Universal Robots URScript: Step Corner Extended.script

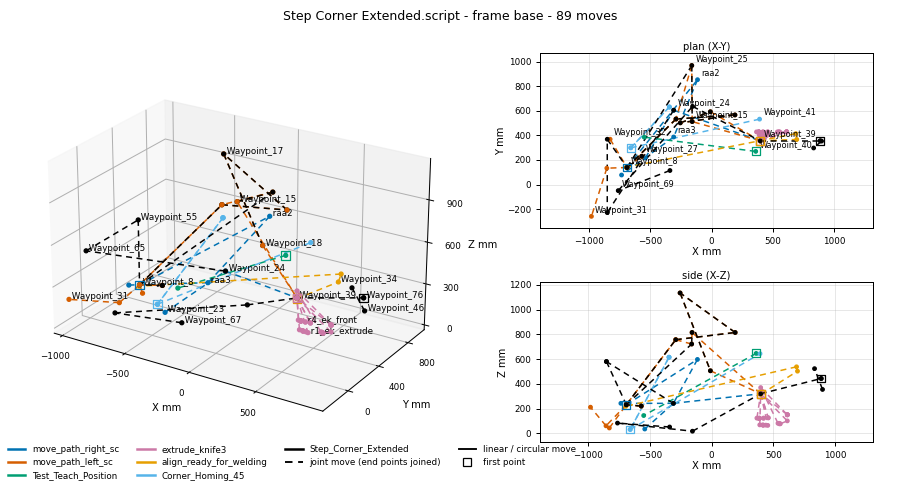
[picture p0: tool path of Step Corner Extended.script in frame base, 89 of 174 moves have a stored position in this frame; points joined in program order, loops and branches not executed]
def Step_Corner_Extended():
  global _hidden_verificationVariable=0
  set_standard_analog_input_domain(0, 1)
  set_standard_analog_input_domain(1, 1)
  set_tool_analog_input_domain(0, 1)
  set_tool_analog_input_domain(1, 1)
  set_analog_outputdomain(0, 0)
  set_analog_outputdomain(1, 0)
  set_input_actions_to_default()
  set_target_payload(10.800000, [-0.001000, -0.053000, 0.068000], [0.081228, 0.081228, 0.081228, 0.000000, 0.000000, 0.000000])
  set_tool_communication(False, 115200, 0, 1, 1.5, 3.5)
  set_tool_output_mode(0)
  set_tool_digital_output_mode(0, 1)
  set_tool_digital_output_mode(1, 1)
  set_tool_voltage(0)
  set_tcp(p[-0.011699999999999999,-0.328,0.105,1.2092,-1.2092,1.2092])
  set_safety_mode_transition_hardness(1)
  set_gravity([0.0, 0.0, 9.82])
  global robot_number=3
  global Point_1=p[0.0,0.0,0.0,0.0,0.0,0.0]
  global Point_2=p[0.0,0.0,0.0,0.0,0.0,0.0]
  # begin: URCap Installation Node
  #   Source: UR Connect, 1.13.79, Universal Robots
  #   Type: UR Connect
  myurRPC = rpc_factory("xmlrpc","http://127.0.0.1:40474")
  # end: URCap Installation Node
  # begin: URCap Installation Node
  #   Source: MachineLogic for Universal Robots, 3.1.7, Vention Inc.
  #   Type: MachineLogic for Universal Robots
  def waitForResponse(expected_response_vention, cname_vention):
  response_vention = socket_read_string(cname_vention,timeout=15)
  while response_vention != expected_response_vention:
  sleep(0.01)
  response_vention = socket_read_string(cname_vention,timeout=15)
  end
  sleep(0.01)
  sync()
  end
  def sendString(string_vention, expected_response_vention, cname_vention):
  socket_send_string(str_cat(string_vention,";"), cname_vention)
  response_vention = socket_read_string(cname_vention,timeout=15)
  if(response_vention == "nAck"):
  popup("nAck received")
  end
  while response_vention != expected_response_vention:
  sleep(0.01)
  response_vention = socket_read_string(cname_vention,timeout=15)
  if(response_vention == "nAck"):
  popup("nAck received")
  end
  end
  sleep(0.01)
  sync()
  end
  def sendStringNAck(string_vention, expected_response_vention, cname_vention):
  socket_send_string(str_cat(string_vention,";"), cname_vention)
  response_vention = socket_read_string(cname_vention,timeout=15)
  if(response_vention == "nAck"):
  popup("nAck received")
  end
  while(response_vention != expected_response_vention and response_vention != "nAck"):
  sleep(0.01)
  response_vention = socket_read_string(cname_vention,timeout=15)
  if(response_vention == "nAck"):
  popup("nAck received",blocking=True)
  end
  end
  sleep(0.01)
  sync()
  end
  def sendStringWithTimeout(string_vention, expected_response_vention, cname_vention):
  socket_send_string(str_cat(string_vention,";"), cname_vention)
  response_vention = socket_read_string(cname_vention,timeout=10)
  if(response_vention == "nAck"):
  popup("nAck received"+string_vention)
  end
  sleep(0.01)
  sync()
  end
  def pollString(string_vention, expected_response_vention, cname_vention):
  socket_send_string(str_cat(string_vention,";"), cname_vention)
  response_vention = socket_read_string(cname_vention,timeout=15)
  if(response_vention == "nAck"):
  popup("nAck received")
  end
  while response_vention != expected_response_vention:
  sleep(1)
  socket_send_string(str_cat(string_vention,";"), cname_vention)
  response_vention = socket_read_string(cname_vention,timeout=15)
  if(response_vention == "nAck"):
  popup("nAck received")
  end
  end
  sleep(0.01)
  sync()
  end
  def sendVariable(var_vention, data_vention, expected_response_vention, cname_vention):
  socket_set_var(var_vention, data_vention, cname_vention)
  response_vention = socket_read_string(cname_vention,timeout=15)
  if(response_vention == "nAck"):
  popup("nAck received")
  end
  while response_vention != expected_response_vention:
  sleep(0.01)
  response_vention = socket_read_string(cname_vention,timeout=15)
  if(response_vention == "nAck"):
  popup("nAck received")
  end
  end
  sleep(0.01)
  sync()
  end
  def intToString(integer_vention,cname_vention):
  stringFix=""
  multiplier_vention123=1
  if integer_vention<0:
  stringFix="-"
  multiplier_vention123=-1
  end
  socket_set_var("GetString",integer_vention*multiplier_vention123,cname_vention)
  string_vention=""
  while string_vention=="":
  sleep(0.01)
  string_vention=socket_read_string(cname_vention,timeout=15)
  end
  sleep(0.01)
  sync()
  string_vention=stringFix+string_vention
  return string_vention
  end
  string_vention=""
  isVentionMovementBusy = False
  isVentionParallelMovementSendingScript = False
  ventionThreadHandle = 1
  isVentionMovementBusyMachineMotion1 = False
  isVentionParallelMovementSendingScriptMachineMotion1 = False
  socket_vention = socket_open("192.168.3.52", 9999, "MachineMotion1")
  if socket_vention==False:
  popup("Check configuration, can't connect to MachineMotion")
  end
  waitForResponse("MachineMotion connection established", "MachineMotion1")
  sendString("isReady", "MachineMotion isReady = true", "MachineMotion1")
  sendStringWithTimeout("setURCapVersion2", "setURCapVersion loaded", "MachineMotion1")
  sendString("SET speed_v2 1000000", "Ack", "MachineMotion1")
  sendString("SET acceleration_v2 100000", "Ack", "MachineMotion1")
  sendString("SET de_axis_1_microsteps_config 8", "Ack", "MachineMotion1")
  sendString("SET de_axis_1_mechanical_gain_config_v2 150000.0", "Ack", "MachineMotion1")
  sendString("SET de_axis_1_direction_config 1", "Ack", "MachineMotion1")
  sendString("SET de_axis_1_type_config Custom Actuator ", "Ack", "MachineMotion1")
  sendString("de_axis_1_config_exec", "Ack", "MachineMotion1")
  # end: URCap Installation Node
  # begin: URCap Installation Node
  #   Source: WireTank Serial, 4.9.0, WireTank, LLC
  #   Type: WireTank Serial
  WTSerialBridge = rpc_factory("xmlrpc","http://127.0.0.1:40511/RPC2")
  # end: URCap Installation Node
  step_count_93fcdbb1_1181_43ea_a7f0_580262fe9a13 = 0.0
  thread Step_Counter_Thread_773b6cc1_d8f8_46f9_9db1_b39c1ae6633a():
    while (True):
      step_count_93fcdbb1_1181_43ea_a7f0_580262fe9a13 = step_count_93fcdbb1_1181_43ea_a7f0_580262fe9a13 + 1.0
      sync()
    end
  end
  run Step_Counter_Thread_773b6cc1_d8f8_46f9_9db1_b39c1ae6633a()
  global free_dr_already=  False
  global freedrive_m_var=  False
  global Waypoint_76_p=p[.886939072471, .356263001241, .442999104957, 2.316306590719, 2.057646408592, .074101958719]
  global Waypoint_76_q=[-3.2647881984118814, -1.2522049299371645, 1.5824044773896437, 0.9175786249801816, -0.008369636028316307, -1.3112608249927966]
  global Waypoint_50_p=p[-.568711442653, .230601791901, .220208834751, -1.519093932087, -.535128035721, .573965472012]
  global Waypoint_50_q=[-0.021522347127095998, -1.2794721287539979, 2.4323821703540247, 5.090870934515753, -2.2996109167682093, 1.533644199371338]
  global Waypoint_51_p=p[-.689649894186, .139001107022, .230693120258, -.852023156701, -1.645963115617, 1.645984943001]
  global Waypoint_51_q=[-1.1454814116107386, -1.5427037247321387, 2.8454700152026575, 4.979047852545538, -4.902958456669943, 1.5718834400177002]
  global Waypoint_52_p=p[-.160992057407, .970528182050, .722037363514, -.554955923310, .106486629259, .328544950173]
  global Waypoint_52_q=[-1.2978580633746546, -1.3217003357461472, 2.2583277861224573, 3.7025129038044433, -2.952825371419088, 0.9627944231033325]
  global Waypoint_53_p=p[-.157624488365, .513351401913, .815670293526, -.672704566373, -1.852329693545, -.055423312366]
  global Waypoint_53_q=[-2.7676661650287073, -1.8206430874266566, 2.312763277684347, 1.0122546392628173, -1.0765226523028772, -0.8102834860431116]
  global Waypoint_54_p=p[-.308528116178, .606080777007, .242371251996, -2.133736658076, .349438277129, 2.130953356703]
  global Waypoint_54_q=[-1.9617512861834925, -1.2994225782207032, 2.207935158406393, 0.745708628291748, 1.5955500602722168, 1.41863214969635]
  global Waypoint_65_p=p[-.850299549699, -.229060500451, .580194265918, -.066683564301, -1.566406749139, -.045536147896]
  global Waypoint_65_q=[0.11527767777442932, -1.206728772526123, 2.660132948552267, 3.2525827127644042, -4.69939905801882, -0.18521625200380498]
  global Waypoint_55_p=p[-.850295942693, .369353811615, .580190947871, -.066690142153, -1.566409865149, -.045506050424]
  global Waypoint_55_q=[-0.89636737505068, -1.198587493305542, 2.6061368624316614, 3.3119169908710937, -4.700617257748739, 0.826545238494873]
  global Waypoint_59_p=p[-.689650832419, .138973473550, .230700469426, -.851985360280, -1.645991124348, 1.645990580233]
  global Waypoint_59_q=[-1.1454528013812464, -1.5427289356342335, 2.8454795519458216, 4.979044186859884, -4.902960960065023, 1.5718833208084106]
  global Waypoint_71_p=p[-.289684660393, .534258475721, .757199031184, -.295236718653, -.653013693815, .389426431276]
  global Waypoint_71_q=[-1.3941848913775843, -1.6550847492613734, 2.7336130777942103, 4.156678839320801, -3.798194471989767, 1.7310842275619507]
  global Waypoint_58_p=p[.191120239889, .567518478899, .815512910186, -.135765364935, .396070873472, .208834263225]
  global Waypoint_58_q=[-1.651280705128805, -1.7712346516051234, 2.617981735860006, 3.3066598612019042, -2.656208101903097, 0.8563313484191895]
  global Waypoint_56_p=p[-.254568281661, .502958752129, 1.135400507516, -.261908057482, -.749714619963, 1.349050618455]
  global Waypoint_56_q=[-2.0344861189471644, -1.9012485943236292, 2.469647232686178, 2.2012061315723876, -1.1677187124835413, -0.5094392935382288]
  global Waypoint_57_p=p[-.009221327687, .593713365169, .505808930157, -1.424394189587, -2.344106819810, -.527597949261]
  global Waypoint_57_q=[-2.920837704335348, -1.9932075939574183, 2.3856611887561243, 0.6815890508839111, -0.5688460508929651, -1.1506975332843226]
  global Waypoint_67_p=p[-.339169194335, .114271165560, .051007401747, -.434162127311, 1.872717119498, -1.885153895998]
  global Waypoint_67_q=[-1.410516087208883, -0.9778240484050293, 2.47756010690798, -1.72361483196401, -0.3956816832171839, 1.808600902557373]
  global Waypoint_69_p=p[-.760826542313, -.049762698068, .082649581767, -1.026233921905, -1.612699318499, 1.547123897415]
  global Waypoint_69_q=[-0.22154647508730108, -1.118469015961029, 2.7561236063586634, -1.5568565337783475, -3.851987902318136, 1.559481143951416]
  global Waypoint_70_p=p[-.154414768496, .636923137577, .016979120256, -.302753655748, 1.486961848367, .122240024639]
  global Waypoint_70_q=[-1.1281922499286097, -1.0678585332683106, 2.4290812651263636, -2.7994214497008265, -1.6034835020648401, 1.7401196956634521]
  global Waypoint_49_p=p[.397354147848, .356263001249, .319808682466, 2.316306590727, 2.057646408591, .074101958728]
  global Waypoint_49_q=[-3.4579480330096644, -2.0568953953185023, 2.3266006151782435, -0.2270372670939942, -0.1993797461139124, -0.10534602800478154]
  global Waypoint_75_p=p[.886939072471, .356263001241, .442999104957, 2.316306590719, 2.057646408592, .074101958719]
  global Waypoint_75_q=[-3.2647881984118814, -1.2522049299371645, 1.5824044773896437, 0.9175786249801816, -0.008369636028316307, -1.3112608249927966]
  global Waypoint_46_p=p[.897631799353, .353934909904, .354805178378, 2.318109555057, 2.056931948624, .061383861333]
  global Waypoint_46_q=[-3.2637236754046843, -1.174605057840683, 1.6528332869159141, 1.0000695425220945, -0.0017340818988245132, -1.5358897417550086]
  global Waypoint_20_p=p[.833090611797, .298095916052, .522915034559, -2.069934341898, -1.817090229983, .262480162787]
  global Waypoint_20_q=[-3.3684676667627205, -1.191816195275802, 1.4015747865517827, 0.7519456332104983, -0.12742073350990069, -0.5504001287532203]
  global Waypoint_8_p=p[-.689650873132, .138963273545, .230691387978, -.851994598965, -1.645998530536, 1.646007616333]
  global Waypoint_8_q=[-0.9414032141314905, -1.501500443821289, 2.801856819783346, 4.981602895050802, -4.698942009602682, 1.571649193763733]
  global raa1_p=p[-.689643170661, .139073527807, .230690921608, -.852069296672, -1.645944888292, 1.645881185303]
  global raa1_q=[-1.1455705801593226, -1.5426994071206828, 2.8454588095294397, 4.979022520571508, -4.9029627482043665, 1.5718539953231812]
  global raa2_p=p[-.114157470946, .855108345894, .597477301975, -.505907028801, .325764798924, .388694870300]
  global raa2_q=[-1.2560303846942347, -1.339010552769043, 2.4151175657855433, 3.6540276247211914, -2.7377544085132044, 1.1360299587249756]
  global raa3_p=p[-.308547482234, .387797636904, .242407099860, 1.976327760240, .350206946999, -1.916000398832]
  global raa3_q=[-1.8931763807879847, -1.3096025747111817, 2.212959591542379, 0.7217818933674316, 1.639076590538025, 0.8125834465026855]
  global raa4_p=p[-.733576132099, .077690893520, .242409727900, 1.976419296976, .350069431278, -1.916084616091]
  global raa4_q=[-0.8909156958209437, -1.3431089532426377, 2.273750130330221, 0.7266384798237304, 1.5611975193023682, 1.8127720355987549]
  global Waypoint_23_p=p[-.540166575654, .215949141041, .034631452617, -1.505795438113, 1.057579835594, 1.573514753692]
  global Waypoint_23_q=[-0.46167117754091436, -1.1365486842444916, 2.508885685597555, 0.15223841249432368, 1.4952874183654785, 3.819530963897705]
  global Waypoint_24_p=p[-.308525559537, .606096497354, .242373144855, -2.133742737559, .349425192770, 2.130939839044]
  global Waypoint_24_q=[-1.8709262053119105, -1.2877716285041352, 2.192875687276022, 0.7510036665150146, 1.5878156423568726, 1.5091480016708374]
  global Waypoint_39_p=p[.397377312153, .356253310648, .319810281486, 2.316317670744, 2.057592854035, .074120023159]
  global Waypoint_39_q=[-3.4579551855670374, -2.0568958721556605, 2.3265963236438196, -0.22706706941638188, -0.19935590425600225, -0.10534030595888311]
  global Waypoint_37_p=p[.397366630181, .356258644196, .319813668943, 2.316299214281, 2.057614642521, .074125657910]
  global Waypoint_37_q=[-3.4579508940326136, -2.056904455224508, 2.3265963236438196, -0.2270481151393433, -0.19937020937074834, -0.10535222688783819]
  global Waypoint_15_p=p[-.157621040248, .513353603496, .815677694745, -.672699538592, -1.852318447516, -.055422773001]
  global Waypoint_15_q=[-2.770456854497091, -1.8207680187621058, 2.3065691629992884, 1.0170823770710449, -1.0767205397235315, -0.8071182409869593]
  global Waypoint_25_p=p[-.161036555831, .970524399959, .722042384791, -.554954311189, .106465018540, .328580879483]
  global Waypoint_25_q=[-1.3071630636798304, -1.3366777312806626, 2.2083633581744593, 3.7187773424335937, -2.9519384543048304, 0.9132363796234131]
  global Waypoint_72_p=p[-.289685725237, .534256396594, .757196155975, -.295237726329, -.653009715205, .389435972469]
  global Waypoint_72_q=[-1.394179646168844, -1.6550847492613734, 2.7336154619800013, 4.156686468715332, -3.7981911341296595, 1.731092095375061]
  global Waypoint_26_p=p[-.689650873132, .138963273545, .230691387978, -.851994598965, -1.645998530536, 1.646007616333]
  global Waypoint_26_q=[-0.9414032141314905, -1.501500443821289, 2.801856819783346, 4.981602895050802, -4.698942009602682, 1.571649193763733]
  global Waypoint_27_p=p[-.568724745609, .230601805298, .220208295176, -1.519097711196, -.535155391172, .573964121010]
  global Waypoint_27_q=[-0.04883271852602178, -1.2753942471793671, 2.4771457354175013, 5.041022258787908, -2.326899592076437, 1.532160997390747]
  global Waypoint_28_p=p[-.568724745609, .230601805298, .220208295176, -1.519097711196, -.535155391172, .573964121010]
  global Waypoint_28_q=[-0.04883271852602178, -1.2753942471793671, 2.4771457354175013, 5.041022258787908, -2.326899592076437, 1.532160997390747]
  global Waypoint_29_p=p[-.689650873132, .138963273545, .230691387978, -.851994598965, -1.645998530536, 1.646007616333]
  global Waypoint_29_q=[-0.9414032141314905, -1.501500443821289, 2.801856819783346, 4.981602895050802, -4.698942009602682, 1.571649193763733]
  global Waypoint_30_p=p[-.853851193668, .133266829906, .060418082908, -.274178222953, -2.359710051999, .046821166283]
  global Waypoint_30_q=[-0.608560864125387, -1.0122360748103638, 2.787060801182882, 3.7283646303364257, -4.940747324620382, 0.3777344226837158]
  global Waypoint_31_p=p[-.979398188272, -.259625449453, .211289397035, -.673010443572, -1.459355862765, -.640164958946]
  global Waypoint_31_q=[0.36968713998794556, -0.5732358259013672, 2.138303581868307, 3.1253925996967773, -4.70385724702944, -1.2100523153888147]
  global Waypoint_32_p=p[-.826865752305, .369357632284, .043113676955, .574997346548, -1.492225541214, .597128135378]
  global Waypoint_32_q=[-1.0355513731585901, -0.33930082738909917, 2.126244846974508, 2.9386045175739746, -4.711197797452108, 1.7860286235809326]
  global Waypoint_33_p=p[-.689650873132, .138963273545, .230691387978, -.851994598965, -1.645998530536, 1.646007616333]
  global Waypoint_33_q=[-0.9414032141314905, -1.501500443821289, 2.801856819783346, 4.981602895050802, -4.698942009602682, 1.571649193763733]
  global Waypoint_73_p=p[-.289671192632, .534275423553, .757232902417, -.295189983811, -.652980753171, .389398176275]
  global Waypoint_73_q=[-1.39418870607485, -1.65509094814443, 2.7335642019854944, 4.156684561366699, -3.7981610933886927, 1.731088399887085]
  global Waypoint_16_p=p[.191112811238, .567512170908, .815514010937, -.135771161622, .396053809900, .208825693369]
  global Waypoint_16_q=[-1.6536315123187464, -1.762029310266012, 2.6225650946246546, 3.2891055780598144, -2.6549678484546106, 0.8520665764808655]
  global Waypoint_17_p=p[-.254565633623, .502963426820, 1.135401557820, -.261910507478, -.749716086887, 1.349041636154]
  global Waypoint_17_q=[-2.035229508076803, -1.8928028545775355, 2.468372408543722, 2.19391576826062, -1.167032543812887, -0.5091407934771937]
  global Waypoint_18_p=p[-.009208376822, .593717720951, .505810027228, -1.424406033077, -2.344120510145, -.527630245278]
  global Waypoint_18_q=[-2.9172328154193323, -1.9945279560484828, 2.3804522196399134, 0.6930715280720214, -0.5671199003802698, -1.1566088835345667]
  global Waypoint_38_p=p[.397379749540, .356252016937, .319817140705, 2.316310534508, 2.057580214841, .074134378577]
  global Waypoint_38_q=[-3.457958761845724, -2.0569073162474574, 2.3265913168536585, -0.22705944002185063, -0.19935638109316045, -0.10534793535341436]
  global Waypoint_40_p=p[.360688403366, .270119715397, .646144746546, .057805349154, 2.125995180379, 2.134053153683]
  global Waypoint_40_q=[-3.4579489866839808, -2.0569035015501917, 2.3265796343432825, -0.22706706941638188, -0.1993501822101038, -0.10534793535341436]
  global Waypoint_2_p=p[-.548957282596, .386284559177, .143710178207, 1.570800598292, -.000025190822, .000004803470]
  global Waypoint_2_q=[-1.0516188780414026, -1.010990933781006, 2.1562450567828577, -1.143702046280243, -1.0526168982135218, -0.0017235914813440445]
  global r1_ek_oldhome_p=p[.397380247322, .356253634699, .319820846021, 2.316316320871, 2.057594704604, .074118471609]
  global r1_ek_oldhome_q=[-3.457949940358297, -2.056894441644186, 2.32658034959902, -0.2270551484874268, -0.19935208955873662, -0.10533696809877569]
  global r1_ek_extrude_p=p[.454852104155, .405448828659, .064015413765, 2.316807606413, 2.051392071696, .076664825947]
  global r1_ek_extrude_q=[-3.274653975163595, -1.5604325172356148, 2.467809502278463, -0.34438879907641606, -0.014281574879781544, -0.6303489843951624]
  global r1_ek_front_p=p[.439064809878, .405452261046, .065996139932, 2.316843937268, 2.051427632497, .076607106393]
  global r1_ek_front_q=[-3.280560557042257, -1.6287623844542445, 2.502561871205465, -0.47416289270434575, -0.019731823598043263, -0.4669149557696741]
  global r1_ek_middle_p=p[.419010105608, .404850828431, .065994665459, 2.309574128677, 2.044678176343, .089098333896]
  global r1_ek_middle_q=[-3.290863100682394, -1.70143522838735, 2.548208538685934, -0.589385525589325, -0.029501263295308888, -0.3372734228717249]
  global r1_ek_middle2_p=p[.417011768852, .405435328663, .065002627117, 2.316867113472, 2.051334925313, .076628493429]
  global r1_ek_middle2_q=[-3.289830032979147, -1.6934038601317347, 2.5445857683764856, -0.579618052845337, -0.028589550648824513, -0.33885270753969365]
  global r1_ek_bottom_p=p[.413071667620, .405431286494, .067999701073, 2.316819721954, 2.051304037200, .076688572349]
  global r1_ek_bottom_q=[-3.2916205565081995, -1.708447118798727, 2.5485368410693567, -0.5849895042232056, -0.03033763567079717, -0.32244998613466436]
  global r1_ek_end_p=p[.389998638281, .405443674081, .068004818811, 2.316851991921, 2.051367741778, .076612018685]
  global r1_ek_end_q=[-3.3030064741717737, -1.7640062771239222, 2.5831297079669397, -0.63420523822818, -0.04154044786562139, -0.2521465460406702]
  global r2_ek_oldhome_p=p[.397380247322, .356253634699, .319820846021, 2.316316320871, 2.057594704604, .074118471609]
  global r2_ek_oldhome_q=[-3.461132842686933, -2.062320779349874, 2.32916033290004, -0.21924456446492258, -0.20097883707844666, -0.11039879152527199]
  global r2_ek_extrude_p=p[.612885745678, .429305279732, .100477107124, 2.149994969793, 2.225764025207, .087353352584]
  global r2_ek_extrude_q=[-3.199475796455825, -1.4862854517875999, 2.263543898005424, -0.6928175084157413, -0.09183293866530295, -0.15653548683830643]
  global r2_ek_front_p=p[.556405415915, .429305279815, .076984362723, -2.170411249256, -2.268200695165, -.015853660170]
  global r2_ek_front_q=[-3.2029012478485694, -1.4943971905029905, 2.3176866046272355, -0.727203417516419, -0.10461513056100813, -0.1013922369747533]
  global r2_ek_middle_p=p[.550033970532, .429305279917, .076253920653, -2.170411249261, -2.268200695170, -.015853660159]
  global r2_ek_middle_q=[-3.2036200175167613, -1.5006788185274456, 2.326226188945654, -0.730095076239345, -0.10533288811000929, -0.10075548926859312]
  global r2_ek_bottom_p=p[.546594660555, .429305280025, .080868477599, -2.170411249265, -2.268200695174, -.015853660149]
  global r2_ek_bottom_q=[-3.204010221105431, -1.5099366263094405, 2.3272215014458872, -0.722096275899732, -0.10572512264357048, -0.10049057923478166]
  global r2_ek_end_p=p[.537335106646, .429305280055, .080868477459, -2.170411249266, -2.268200695175, -.015853660146]
  global r2_ek_end_q=[-3.205098875769389, -1.5204959829395506, 2.3387656715508855, -0.724001524008818, -0.10681294496314919, -0.09956563917089412]
  global r3_ek_oldhome_p=p[.397385850131, .356252441346, .369809999696, 2.316320575836, 2.057576093691, .074125563417]
  global r3_ek_oldhome_q=[-3.4600108097540825, -2.084533794186367, 2.2686976909438377, -0.1444297831854957, -0.20178034518575938, -0.10248789488416588]
  global r3_ek_extrude_p=p[.612883684377, .429310301838, .149999999683, 2.149962295817, 2.225777492182, .087374550826]
  global r3_ek_extrude_q=[-3.1980123446153748, -1.538400201434774, 2.229744902146236, -0.6115506790497731, -0.09278008251792791, -0.15193191663383665]
  global r3_ek_front_p=p[.612883684377, .429310301838, .149999999683, 2.149962295817, 2.225777492182, .087374550826]
  global r3_ek_front_q=[-3.1980123446153748, -1.538400201434774, 2.229744902146236, -0.6115506790497731, -0.09278008251792791, -0.15193191663383665]
  global r3_ek_middle_p=p[.612883684377, .429310301838, .149999999683, 2.149962295817, 2.225777492182, .087374550826]
  global r3_ek_middle_q=[-3.1980123446153748, -1.538400201434774, 2.229744902146236, -0.6115506790497731, -0.09278008251792791, -0.15193191663383665]
  global r3_ek_bottom_p=p[.612883684377, .429310301838, .149999999683, 2.149962295817, 2.225777492182, .087374550826]
  global r3_ek_bottom_q=[-3.1980123446153748, -1.538400201434774, 2.229744902146236, -0.6115506790497731, -0.09278008251792791, -0.15193191663383665]
  global r3_ek_end_p=p[.612883684377, .429310301838, .149999999683, 2.149962295817, 2.225777492182, .087374550826]
  global r3_ek_end_q=[-3.1980123446153748, -1.538400201434774, 2.229744902146236, -0.6115506790497731, -0.09278008251792791, -0.15193191663383665]
  global r4_ek_oldhome_p=p[.397380247322, .356253634699, .319820846021, 2.316316320871, 2.057594704604, .074118471609]
  global r4_ek_oldhome_q=[-3.4680860338785493, -2.070376223306912, 2.3329367157510497, -0.22828162349163783, -0.20619604348947362, -0.09694130604598783]
  global r4_ek_extrude_p=p[.458670548589, .429305279741, .125141489362, 2.149994969793, 2.225764025207, .087353352584]
  global r4_ek_extrude_q=[-3.224306558956634, -1.7135315940479465, 2.43410270276974, -0.6768839938806144, -0.1154143142053492, -0.11562209601533713]
  global r4_ek_front_p=p[.420084046436, .429305279533, .122370065986, -2.206701899775, -2.177374452500, .052747240372]
  global r4_ek_front_q=[-3.2223885287117087, -1.7265329174617632, 2.4434355314143925, -0.6644243149558609, -0.06512925128431313, -0.01659929377642566]
  global r4_ek_middle_p=p[.385663706386, .429305279588, .119862350556, -2.206701899778, -2.177374452500, .052747240377]
  global r4_ek_middle_q=[-3.2295441306515738, -1.774240686665987, 2.4822688267544946, -0.6583601229072489, -0.07232201786773373, -0.0137735297523216]
  global r4_ek_bottom_p=p[.385663706260, .429305279599, .122809894660, -2.206701899778, -2.177374452501, .052747240377]
  global r4_ek_bottom_q=[-3.2295577467539287, -1.7778480193330992, 2.4794176409730713, -0.6518633442593682, -0.07233077879629679, -0.013811892538432069]
  global r4_ek_end_p=p[.366757227289, .429305279628, .122809894538, -2.206701899780, -2.177374452501, .052747240380]
  global r4_ek_end_q=[-3.2341047638544715, -1.8072551968371293, 2.4987903200913473, -0.6435011221874376, -0.07689850609233773, -0.01212997029934737]
  global oldhome_p=p[.397683836105, .356251384911, .315246899233, 2.316304177919, 2.057561756051, .074146544723]
  global oldhome_q=[-3.457960907612936, -2.0569125614561976, 2.326589886342184, -0.22707636774096684, -0.19935208955873662, -0.10534269014467412]
  global Waypoint_34_p=p[.695155464390, .367451880816, .502522491683, 2.093108370749, 1.857548644474, .308841595089]
  global Waypoint_34_q=[-3.249415699635641, -1.9387923679747523, 2.3226097265826624, 3.981850786800049, -0.05697328249086553, 1.5286790132522583]
  global Waypoint_35_p=p[.687527620967, .415165960724, .537921070000, 2.127101811831, 1.929915403723, .470130777221]
  global Waypoint_35_q=[-3.249424997960226, -1.9387947521605433, 2.32263428369631, 3.9818588930317382, -6.198007937763826, 1.5286580324172974]
  global Waypoint_36_p=p[-.693756081485, .141369193308, .218584735520, -.851978179689, -1.646001533937, 1.646008371360]
  global Waypoint_36_q=[-1.1533568541156214, -1.4924076360515137, 2.8518698851214808, 4.922323781042852, -4.910887185727255, 1.5719373226165771]
  def calculate_point_to_move_towards(feature, direction, position_distance):
    local posDir=[direction[0], direction[1], direction[2]]
    if (norm(posDir) < 1e-6):
      return get_target_waypoint()
    end
    local direction_vector_normalized=normalize(posDir)
    local displacement_pose=p[direction_vector_normalized[0] * position_distance,direction_vector_normalized[1] * position_distance,direction_vector_normalized[2] * position_distance,0,0,0]
    local wanted_displacement_in_base_frame=pose_sub(pose_trans(feature, displacement_pose), feature)
    return pose_add(get_target_waypoint(), wanted_displacement_in_base_frame)
  end
  global Waypoint_4_p=p[-.658264763546, .299530128456, .030909835036, .426821001551, -1.621505068649, .437070885767]
  global Waypoint_4_q=[-1.350241486226217, -0.9702387017062684, 2.492185179387228, -1.7834822140135707, -0.33723670641054326, 1.8489984273910522]
  global Waypoint_13_p=p[-.343952006273, .632142227752, .615174722549, -.025948978133, -.008794819136, -.567469912202]
  global Waypoint_13_q=[-1.350241486226217, -0.9702451390079041, 2.492171827946798, -3.0669099293150843, 1.575993537902832, 2.355180025100708]
  global Waypoint_1_p=p[-.343952006258, .632142227456, .615174722551, -.025016780489, .033118613186, -3.068519793995]
  global Waypoint_1_q=[-1.3432858302651205, -0.8819789687502322, 2.478150442072055, -3.1920490209023007, 1.5816449765089289, -0.1549241290366341]
  global Waypoint_14_p=p[-.343952006273, .632142227752, .615174722549, -.025948978133, -.008794819136, -.567469912202]
  global Waypoint_14_q=[-1.350241486226217, -0.9702451390079041, 2.492171827946798, -3.0669099293150843, 1.575993537902832, 2.355180025100708]
  global Waypoint_41_p=p[.392127936214, .533269017847, .644148583936, .057822570580, 2.125982462550, 2.134033989912]
  global Waypoint_41_q=[-3.4579578081714075, -2.0569120846190394, 2.3265841642962855, -0.22706885755572515, -0.1993349234210413, -0.10534984270204717]
  def move_path_right_sc():
    $ 136 "move_path_right_sc" "noBreak"
    $ 137 "'this is the path for Down, Over, then Back Around'"
    # 'this is the path for Down, Over, then Back Around'
    $ 138 "Comment"
    # Comment
    $ 147 "align_ready_for_welding()"
    align_ready_for_welding()
    $ 148 "Comment"
    # Comment
    $ 149 "Set"
    set_tcp(p[-0.011699999999999999,-0.328,0.105,1.2092,-1.2092,1.2092])
    $ 150 "p1≔pathturn[0]"
    global p1=pathturn[0]
    $ 151 "p2≔pathturn[1]"
    global p2=pathturn[1]
    $ 152 "p4≔pathturn[2]"
    global p4=pathturn[2]
    $ 153 "p5≔pathturn[3]"
    global p5=pathturn[3]
    $ 154 "pa1≔p[p1[0]+0.05,p1[1]+0.05,p1[2],p1[3],p1[4],p1[5]]"
    global pa1=p[p1[0]+0.05,p1[1]+0.05,p1[2],p1[3],p1[4],p1[5]]
    $ 155 "p6≔pathturn[9]"
    global p6=pathturn[9]
    $ 156 "p7≔pathturn[10]"
    global p7=pathturn[10]
    $ 157 "p8≔pathturn[11]"
    global p8=pathturn[11]
    $ 158 "liftcolumnup"
    $ 159 "liftcolumnz≔liftcolumnzneeded"
    global liftcolumnz=liftcolumnzneeded
    $ 160 "If liftcolumnz>0"
    if (liftcolumnz>0):
      # begin: URCap Program Node
      #   Source: MachineLogic for Universal Robots, 3.1.7, Vention Inc.
      #   Type: MachineLogic for Universal Robots
      $ 161 "MachineLogic Move to Position"
      while isVentionMovementBusyMachineMotion1==True:
      sleep(0.05)
      end
      if(isVentionMovementBusyMachineMotion1 == False):
      isVentionMovementBusyMachineMotion1 = True
      socket_send_string("estop/status;", "MachineMotion1")
      temp_estop_var_vention = socket_read_string("MachineMotion1",timeout=15)
      while(temp_estop_var_vention=="estop/status true"):
      if temp_estop_var_vention=="estop/status true":
      sendStringWithTimeout("estop/systemreset/request","Ack estop/systemreset/request;","MachineMotion1")
      end
      socket_send_string("estop/status;", "MachineMotion1")
      temp_estop_var_vention = socket_read_string("MachineMotion1",timeout=15)
      if temp_estop_var_vention=="estop/status true":
      popup("MachineMotion in estop, make sure you have all emergency modules released manually. If you continue the system will try to reset MachineMotion automatically.",blocking=True)
      end
      end
      else:
      popup("resource is being used already: MachineMotion1")
      halt
      end
      sendString("SET speed_v2 3000000.000", "Ack", "MachineMotion1")
      sendString("SET acceleration_v2 50000.000", "Ack", "MachineMotion1")
      string_vention=intToString(liftcolumnz*1000,"MachineMotion1")
      sendString("SET de_move_abs_1 "+string_vention, "Ack", "MachineMotion1")
      sendString("de_move_abs_exec", "Ack", "MachineMotion1")
      isVentionParallelMovementSendingScriptMachineMotion1 = False
      pollString("isMotionCompleted", "MachineMotion isMotionCompleted = true", "MachineMotion1")
      isVentionMovementBusyMachineMotion1 = False
      sleep(0.03)
      # end: URCap Program Node
    end
    $ 162 "MoveJ"
    $ 163 "pa1" "breakAfter"
    movej(pa1, a=1.3962634015954636, v=0.3490658503988659)
    $ 164 "MoveL"
    $ 165 "p1" "breakAfter"
    movel(p1, a=0.2, v=0.05)
    $ 166 "Wait: 8.0"
    sleep(8.0)
    # begin: URCap Program Node
    #   Source: WireTank Serial, 4.9.0, WireTank, LLC
    #   Type: WireTank Serial
    $ 167 "Serial Bridge uR1"
    SerialResponse = WTSerialBridge.send_command("/dev/ttyUSB0",1200, 8, "None", "One", "None", 1000, "None", "None", [252,82,49], False)
    # end: URCap Program Node
    # begin: URCap Program Node
    #   Source: WireTank Serial, 4.9.0, WireTank, LLC
    #   Type: WireTank Serial
    $ 168 "Serial Bridge uR1"
    SerialResponse = WTSerialBridge.send_command("/dev/ttyUSB0",1200, 8, "None", "One", "None", 1000, "None", "None", [252,82,49], False)
    # end: URCap Program Node
    $ 169 "Wait: 1.0"
    sleep(1.0)
    $ 171 "Set DO[0]=On"
    set_standard_digital_out(0, True)
    $ 172 "MoveL"
    $ 173 "p2" "breakAfter"
    movel(p2, a=0.1, v=0.01)
    # begin: URCap Program Node
    #   Source: WireTank Serial, 4.9.0, WireTank, LLC
    #   Type: WireTank Serial
    $ 174 "Serial Bridge uR0"
    SerialResponse = WTSerialBridge.send_command("/dev/ttyUSB0",1200, 8, "None", "One", "None", 1000, "None", "None", [252,82,48], False)
    # end: URCap Program Node
    $ 175 "Wait: 0.5"
    sleep(0.5)
    $ 176 "Set DO[0]=Off"
    set_standard_digital_out(0, False)
    $ 177 "MoveL"
    $ 178 "p4" "breakAfter"
    movel(p4, a=0.01, v=0.12)
    # begin: URCap Program Node
    #   Source: WireTank Serial, 4.9.0, WireTank, LLC
    #   Type: WireTank Serial
    $ 179 "Serial Bridge uR1"
    SerialResponse = WTSerialBridge.send_command("/dev/ttyUSB0",1200, 8, "None", "One", "None", 1000, "None", "None", [252,82,49], False)
    # end: URCap Program Node
    # begin: URCap Program Node
    #   Source: WireTank Serial, 4.9.0, WireTank, LLC
    #   Type: WireTank Serial
    $ 180 "Serial Bridge uR1"
    SerialResponse = WTSerialBridge.send_command("/dev/ttyUSB0",1200, 8, "None", "One", "None", 1000, "None", "None", [252,82,49], False)
    # end: URCap Program Node
    $ 181 "Wait: 1.0"
    sleep(1.0)
    $ 183 "Set DO[0]=On"
    set_standard_digital_out(0, True)
    $ 184 "MoveL"
    $ 186 "p6" "breakAfter"
    movel(p6, a=0.1, v=0.01)
    $ 187 "p7" "breakAfter"
    movel(p7, a=0.1, v=0.01)
    # begin: URCap Program Node
    #   Source: WireTank Serial, 4.9.0, WireTank, LLC
    #   Type: WireTank Serial
    $ 188 "Serial Bridge uR0"
    SerialResponse = WTSerialBridge.send_command("/dev/ttyUSB0",1200, 8, "None", "One", "None", 1000, "None", "None", [252,82,48], False)
    # end: URCap Program Node
    $ 189 "Set DO[0]=Off"
    set_standard_digital_out(0, False)
    $ 190 "MoveL"
    $ 191 "p8" "breakAfter"
    movel(p8, a=0.1, v=0.01)
    $ 193 "Set DO[0]=Off"
    set_standard_digital_out(0, False)
    $ 194 "Comment"
    # Comment
    $ 195 "pret1≔p[p5[0]+.1,p5[1],p5[2],p5[3],p5[4],p5[5]]"
    global pret1=p[p5[0]+.1,p5[1],p5[2],p5[3],p5[4],p5[5]]
    $ 196 "p_1≔pathturn[4]"
    global p_1=pathturn[4]
    $ 197 "p_2≔pathturn[5]"
    global p_2=pathturn[5]
    $ 198 "p_3≔pathturn[6]"
    global p_3=pathturn[6]
    $ 199 "p_4≔pathturn[7]"
    global p_4=pathturn[7]
    $ 200 "p_5≔pathturn[8]"
    global p_5=pathturn[8]
    $ 201 "p_preheat≔p[p_3[0]+.01,p_3[1],p_3[2],p_3[3],p_3[4],p_3[5]]"
    global p_preheat=p[p_3[0]+.01,p_3[1],p_3[2],p_3[3],p_3[4],p_3[5]]
    $ 202 "p_pre_ret≔p[p_1[0]+.03,p_1[1]+.03,p_1[2],p_1[3],p_1[4],p_1[5]]"
    global p_pre_ret=p[p_1[0]+.03,p_1[1]+.03,p_1[2],p_1[3],p_1[4],p_1[5]]
    $ 203 "p_pre_ret2≔p[p_3[0]+.1,p_3[1],p_3[2],p_3[3],p_3[4],p_3[5]]"
    global p_pre_ret2=p[p_3[0]+.1,p_3[1],p_3[2],p_3[3],p_3[4],p_3[5]]
    $ 204 "p_6≔pathturn[12]"
    global p_6=pathturn[12]
    $ 205 "p_7≔pathturn[13]"
    global p_7=pathturn[13]
    $ 206 "p_8≔pathturn[14]"
    global p_8=pathturn[14]
    $ 207 "'twist'"
    # 'twist'
    $ 208 "MoveJ"
    $ 209 "pret1" "breakAfter"
    movej(pret1, a=1.3962634015954636, v=1.3962634015954636)
    $ 210 "Waypoint_8" "breakAfter"
    movej(get_inverse_kin(Waypoint_8_p, qnear=Waypoint_8_q), a=1.3962634015954636, v=1.0471975511965976)
    $ 212 "MoveJ"
    $ 213 "raa1" "breakAfter"
    movej(get_inverse_kin(raa1_p, qnear=raa1_q), a=1.3962634015954636, v=1.0471975511965976)
    $ 214 "raa2" "breakAfter"
    movej(get_inverse_kin(raa2_p, qnear=raa2_q), a=1.3962634015954636, v=1.0471975511965976)
    $ 215 "raa3" "breakAfter"
    movej(get_inverse_kin(raa3_p, qnear=raa3_q), a=1.3962634015954636, v=1.0471975511965976)
    $ 216 "raa4" "breakAfter"
    movej(get_inverse_kin(raa4_p, qnear=raa4_q), a=1.3962634015954636, v=1.0471975511965976)
    $ 218 "If liftcolumnz≠0.0"
    if (liftcolumnz != 0.0):
      # begin: URCap Program Node
      #   Source: MachineLogic for Universal Robots, 3.1.7, Vention Inc.
      #   Type: MachineLogic for Universal Robots
      $ 219 "MachineLogic Homing"
      while isVentionMovementBusyMachineMotion1==True:
      sleep(0.05)
      end
      if(isVentionMovementBusyMachineMotion1 == False):
      isVentionMovementBusyMachineMotion1 = True
      socket_send_string("estop/status;", "MachineMotion1")
      temp_estop_var_vention = socket_read_string("MachineMotion1",timeout=15)
      while(temp_estop_var_vention=="estop/status true"):
      if temp_estop_var_vention=="estop/status true":
      sendStringWithTimeout("estop/systemreset/request","Ack estop/systemreset/request;","MachineMotion1")
      end
      socket_send_string("estop/status;", "MachineMotion1")
      temp_estop_var_vention = socket_read_string("MachineMotion1",timeout=15)
      if temp_estop_var_vention=="estop/status true":
      popup("MachineMotion in estop, make sure you have all emergency modules released manually. If you continue the system will try to reset MachineMotion automatically.",blocking=True)
      end
      end
      else:
      popup("resource is being used already: MachineMotion1")
      halt
      end
      isVentionMovementBusyMachineMotion1 = True
      sendString("im_home_axis_1", "MachineMotion im_home_axis_1 = completed", "MachineMotion1")
      isVentionMovementBusyMachineMotion1 = False
      sendString("SET im_set_encoder_pos_aux_1 0.000", "Ack", "MachineMotion1")
      isVentionMovementBusyMachineMotion1 = False
      sleep(0.03)
      # end: URCap Program Node
    end
    $ 220 "'preheat'"
    # 'preheat'
    $ 223 "MoveL"
    $ 224 "p_pre_ret2" "breakAfter"
    movel(p_pre_ret2, a=1.2, v=0.25)
    $ 225 "p_preheat" "breakAfter"
    movel(p_preheat, a=1.2, v=0.25)
    $ 226 "Wait: 6.0"
    sleep(6.0)
    $ 227 "MoveL"
    $ 228 "p_pre_ret2" "breakAfter"
    movel(p_pre_ret2, a=1.2, v=0.25)
    $ 229 "p_pre_ret" "breakAfter"
    movel(p_pre_ret, a=1.2, v=0.25)
    $ 230 "Set"
    set_tcp(p[0.00451,-0.328,0.105,1.2092,-1.2092,1.2092])
    $ 231 "MoveL"
    $ 232 "p_1" "breakAfter"
    movel(p_1, a=1.2, v=0.05)
    # begin: URCap Program Node
    #   Source: WireTank Serial, 4.9.0, WireTank, LLC
    #   Type: WireTank Serial
    $ 233 "Serial Bridge uR1"
    SerialResponse = WTSerialBridge.send_command("/dev/ttyUSB0",1200, 8, "None", "One", "None", 1000, "None", "None", [252,82,49], False)
    # end: URCap Program Node
    # begin: URCap Program Node
    #   Source: WireTank Serial, 4.9.0, WireTank, LLC
    #   Type: WireTank Serial
    $ 234 "Serial Bridge uR1"
    SerialResponse = WTSerialBridge.send_command("/dev/ttyUSB0",1200, 8, "None", "One", "None", 1000, "None", "None", [252,82,49], False)
    # end: URCap Program Node
    $ 235 "Wait: 1.0"
    sleep(1.0)
    $ 236 "Set DO[0]=On"
    set_standard_digital_out(0, True)
    $ 238 "Wait: 1.0"
    sleep(1.0)
    $ 239 "MoveL"
    $ 240 "p_2" "breakAfter"
    movel(p_2, a=1.2, v=0.01)
    $ 241 "MoveP"
    $ 242 "CircleMove"
    $ 243 "p_3" "noBreak"

    $ 244 "p_4" "breakAfter"
    movec(p_3, p_4, a=0.01, v=5.0E-4, r=0.0, mode=1)
    $ 245 "MoveL"
    $ 246 "p_5" "breakAfter"
    movel(p_5, a=1.2, v=0.012)
    $ 247 "Set"
    set_tcp(p[-0.011699999999999999,-0.328,0.105,1.2092,-1.2092,1.2092])
    $ 248 "MoveL"
    $ 249 "p_6" "breakAfter"
    movel(p_6, a=0.1, v=0.012)
    $ 250 "p_7" "breakAfter"
    movel(p_7, a=0.1, v=0.012)
    # begin: URCap Program Node
    #   Source: WireTank Serial, 4.9.0, WireTank, LLC
    #   Type: WireTank Serial
    $ 251 "Serial Bridge uR0"
    SerialResponse = WTSerialBridge.send_command("/dev/ttyUSB0",1200, 8, "None", "One", "None", 1000, "None", "None", [252,82,48], False)
    # end: URCap Program Node
    $ 252 "Set DO[0]=Off"
    set_standard_digital_out(0, False)
    $ 254 "MoveL"
    $ 255 "p_8" "breakAfter"
    movel(p_8, a=0.1, v=0.01)
    $ 256 "Set DO[0]=Off"
    set_standard_digital_out(0, False)
    $ 257 "MoveL"
    $ 258 "Waypoint_23" "breakAfter"
    movel(Waypoint_23_p, a=1.2, v=0.25)
    $ 259 "MoveJ"
    $ 260 "Waypoint_24" "breakAfter"
    movej(get_inverse_kin(Waypoint_24_p, qnear=Waypoint_24_q), a=1.3962634015954636, v=1.0471975511965976)
    $ 261 "Waypoint_39" "breakAfter"
    movej(get_inverse_kin(Waypoint_39_p, qnear=Waypoint_39_q), a=1.3962634015954636, v=1.0471975511965976)
    $ 262 "'above waypoint is home'"
    # 'above waypoint is home'
  end
  def move_path_left_sc():
    $ 263 "move_path_left_sc" "noBreak"
    $ 264 "'this is the path for Down, Over, then Back Around'"
    # 'this is the path for Down, Over, then Back Around'
    $ 265 "Comment"
    # Comment
    $ 266 "MoveJ"
    $ 267 "Waypoint_37" "breakAfter"
    movej(get_inverse_kin(Waypoint_37_p, qnear=Waypoint_37_q), a=1.3962634015954636, v=1.0471975511965976)
    $ 268 "'above point is home'"
    # 'above point is home'
    $ 269 "liftcolumnup"
    $ 270 "liftcolumnz≔liftcolumnzneeded"
    global liftcolumnz=liftcolumnzneeded
    $ 271 "If liftcolumnz>0"
    if (liftcolumnz>0):
      # begin: URCap Program Node
      #   Source: MachineLogic for Universal Robots, 3.1.7, Vention Inc.
      #   Type: MachineLogic for Universal Robots
      $ 272 "MachineLogic Move to Position"
      while isVentionMovementBusyMachineMotion1==True:
      sleep(0.05)
      end
      if(isVentionMovementBusyMachineMotion1 == False):
      isVentionMovementBusyMachineMotion1 = True
      socket_send_string("estop/status;", "MachineMotion1")
      temp_estop_var_vention = socket_read_string("MachineMotion1",timeout=15)
      while(temp_estop_var_vention=="estop/status true"):
      if temp_estop_var_vention=="estop/status true":
      sendStringWithTimeout("estop/systemreset/request","Ack estop/systemreset/request;","MachineMotion1")
      end
      socket_send_string("estop/status;", "MachineMotion1")
      temp_estop_var_vention = socket_read_string("MachineMotion1",timeout=15)
      if temp_estop_var_vention=="estop/status true":
      popup("MachineMotion in estop, make sure you have all emergency modules released manually. If you continue the system will try to reset MachineMotion automatically.",blocking=True)
      end
      end
      else:
      popup("resource is being used already: MachineMotion1")
      halt
      end
      sendString("SET speed_v2 3000000.000", "Ack", "MachineMotion1")
      sendString("SET acceleration_v2 50000.000", "Ack", "MachineMotion1")
      string_vention=intToString(liftcolumnz*1000,"MachineMotion1")
      sendString("SET de_move_abs_1 "+string_vention, "Ack", "MachineMotion1")
      sendString("de_move_abs_exec", "Ack", "MachineMotion1")
      isVentionParallelMovementSendingScriptMachineMotion1 = False
      pollString("isMotionCompleted", "MachineMotion isMotionCompleted = true", "MachineMotion1")
      isVentionMovementBusyMachineMotion1 = False
      sleep(0.03)
      # end: URCap Program Node
    end
    $ 273 "Waypoint_15" "breakAfter"
    movej(get_inverse_kin(Waypoint_15_p, qnear=Waypoint_15_q), a=1.3962634015954636, v=1.0471975511965976)
    $ 274 "Waypoint_25" "breakAfter"
    movej(get_inverse_kin(Waypoint_25_p, qnear=Waypoint_25_q), a=1.3962634015954636, v=1.0471975511965976)
    $ 275 "Waypoint_72" "breakAfter"
    movej(get_inverse_kin(Waypoint_72_p, qnear=Waypoint_72_q), a=1.3962634015954636, v=1.0471975511965976)
    $ 276 "Waypoint_26" "breakAfter"
    movej(get_inverse_kin(Waypoint_26_p, qnear=Waypoint_26_q), a=1.3962634015954636, v=1.0471975511965976)
    $ 277 "Waypoint_27" "breakAfter"
    movej(get_inverse_kin(Waypoint_27_p, qnear=Waypoint_27_q), a=1.3962634015954636, v=1.0471975511965976)
    $ 282 "Comment"
    # Comment
    $ 283 "Set"
    set_tcp(p[-0.011699999999999999,-0.328,0.105,1.2092,-1.2092,1.2092])
    $ 284 "p1≔pathturn[0]"
    global p1=pathturn[0]
    $ 285 "p2≔pathturn[1]"
    global p2=pathturn[1]
    $ 286 "p4≔pathturn[2]"
    global p4=pathturn[2]
    $ 287 "p5≔pathturn[3]"
    global p5=pathturn[3]
    $ 288 "pa1≔p[p1[0]+0.05,p1[1]-0.05,p1[2],p1[3],p1[4],p1[5]]"
    global pa1=p[p1[0]+0.05,p1[1]-0.05,p1[2],p1[3],p1[4],p1[5]]
    $ 289 "p6≔pathturn[9]"
    global p6=pathturn[9]
    $ 290 "p7≔pathturn[10]"
    global p7=pathturn[10]
    $ 291 "p8≔pathturn[11]"
    global p8=pathturn[11]
    $ 292 "MoveJ"
    $ 293 "pa1" "breakAfter"
    movej(pa1, a=1.3962634015954636, v=1.0471975511965976)
    $ 294 "MoveL"
    $ 295 "p1" "breakAfter"
    movel(p1, a=0.1, v=0.05)
    $ 296 "Wait: 8.0"
    sleep(8.0)
    # begin: URCap Program Node
    #   Source: WireTank Serial, 4.9.0, WireTank, LLC
    #   Type: WireTank Serial
    $ 297 "Serial Bridge uR1"
    SerialResponse = WTSerialBridge.send_command("/dev/ttyUSB0",1200, 8, "None", "One", "None", 1000, "None", "None", [252,82,49], False)
    # end: URCap Program Node
    # begin: URCap Program Node
    #   Source: WireTank Serial, 4.9.0, WireTank, LLC
    #   Type: WireTank Serial
    $ 298 "Serial Bridge uR1"
    SerialResponse = WTSerialBridge.send_command("/dev/ttyUSB0",1200, 8, "None", "One", "None", 1000, "None", "None", [252,82,49], False)
    # end: URCap Program Node
    $ 299 "Wait: 1.0"
    sleep(1.0)
    $ 301 "Set DO[0]=On"
    set_standard_digital_out(0, True)
    $ 302 "MoveL"
    $ 303 "p2" "breakAfter"
    movel(p2, a=0.1, v=0.01)
    # begin: URCap Program Node
    #   Source: WireTank Serial, 4.9.0, WireTank, LLC
    #   Type: WireTank Serial
    $ 304 "Serial Bridge uR0"
    SerialResponse = WTSerialBridge.send_command("/dev/ttyUSB0",1200, 8, "None", "One", "None", 1000, "None", "None", [252,82,48], False)
    # end: URCap Program Node
    $ 305 "Wait: 0.5"
    sleep(0.5)
    $ 306 "Set DO[0]=Off"
    set_standard_digital_out(0, False)
    $ 307 "MoveL"
    $ 308 "p4" "breakAfter"
    movel(p4, a=0.01, v=0.12)
    # begin: URCap Program Node
    #   Source: WireTank Serial, 4.9.0, WireTank, LLC
    #   Type: WireTank Serial
    $ 309 "Serial Bridge uR1"
    SerialResponse = WTSerialBridge.send_command("/dev/ttyUSB0",1200, 8, "None", "One", "None", 1000, "None", "None", [252,82,49], False)
    # end: URCap Program Node
    # begin: URCap Program Node
    #   Source: WireTank Serial, 4.9.0, WireTank, LLC
    #   Type: WireTank Serial
    $ 310 "Serial Bridge uR1"
    SerialResponse = WTSerialBridge.send_command("/dev/ttyUSB0",1200, 8, "None", "One", "None", 1000, "None", "None", [252,82,49], False)
    # end: URCap Program Node
    $ 311 "Wait: 1.0"
    sleep(1.0)
    $ 313 "Set DO[0]=On"
    set_standard_digital_out(0, True)
    $ 314 "MoveL"
    $ 316 "p6" "breakAfter"
    movel(p6, a=0.1, v=0.01)
    $ 317 "p7" "breakAfter"
    movel(p7, a=0.1, v=0.01)
    # begin: URCap Program Node
    #   Source: WireTank Serial, 4.9.0, WireTank, LLC
    #   Type: WireTank Serial
    $ 318 "Serial Bridge uR0"
    SerialResponse = WTSerialBridge.send_command("/dev/ttyUSB0",1200, 8, "None", "One", "None", 1000, "None", "None", [252,82,48], False)
    # end: URCap Program Node
    $ 319 "Set DO[0]=Off"
    set_standard_digital_out(0, False)
    $ 320 "MoveL"
    $ 321 "p8" "breakAfter"
    movel(p8, a=0.1, v=0.01)
    $ 323 "Set DO[0]=Off"
    set_standard_digital_out(0, False)
    $ 324 "Comment"
    # Comment
    $ 325 "pret1≔p[p5[0]+.1,p5[1],p5[2],p5[3],p5[4],p5[5]]"
    global pret1=p[p5[0]+.1,p5[1],p5[2],p5[3],p5[4],p5[5]]
    $ 326 "p_1≔pathturn[4]"
    global p_1=pathturn[4]
    $ 327 "p_2≔pathturn[5]"
    global p_2=pathturn[5]
    $ 328 "p_3≔pathturn[6]"
    global p_3=pathturn[6]
    $ 329 "p_4≔pathturn[7]"
    global p_4=pathturn[7]
    $ 330 "p_5≔pathturn[8]"
    global p_5=pathturn[8]
    $ 331 "p_preheat≔p[p_3[0]+.01,p_3[1],p_3[2],p_3[3],p_3[4],p_3[5]]"
    global p_preheat=p[p_3[0]+.01,p_3[1],p_3[2],p_3[3],p_3[4],p_3[5]]
    $ 332 "p_pre_ret≔p[p_1[0]+.03,p_1[1]-.03,p_1[2],p_1[3],p_1[4],p_1[5]]"
    global p_pre_ret=p[p_1[0]+.03,p_1[1]-.03,p_1[2],p_1[3],p_1[4],p_1[5]]
    $ 333 "p_pre_ret2≔p[p_3[0]+.03,p_3[1],p_3[2],p_3[3],p_3[4],p_3[5]]"
    global p_pre_ret2=p[p_3[0]+.03,p_3[1],p_3[2],p_3[3],p_3[4],p_3[5]]
    $ 334 "p_6≔pathturn[12]"
    global p_6=pathturn[12]
    $ 335 "p_7≔pathturn[13]"
    global p_7=pathturn[13]
    $ 336 "p_8≔pathturn[14]"
    global p_8=pathturn[14]
    $ 337 "MoveJ"
    $ 338 "pret1" "breakAfter"
    movej(pret1, a=1.3962634015954636, v=1.3962634015954636)
    $ 339 "Waypoint_28" "breakAfter"
    movej(get_inverse_kin(Waypoint_28_p, qnear=Waypoint_28_q), a=1.3962634015954636, v=1.3962634015954636)
    $ 340 "If liftcolumnz≠0.0"
    if (liftcolumnz != 0.0):
      # begin: URCap Program Node
      #   Source: MachineLogic for Universal Robots, 3.1.7, Vention Inc.
      #   Type: MachineLogic for Universal Robots
      $ 341 "MachineLogic Homing"
      while isVentionMovementBusyMachineMotion1==True:
      sleep(0.05)
      end
      if(isVentionMovementBusyMachineMotion1 == False):
      isVentionMovementBusyMachineMotion1 = True
      socket_send_string("estop/status;", "MachineMotion1")
      temp_estop_var_vention = socket_read_string("MachineMotion1",timeout=15)
      while(temp_estop_var_vention=="estop/status true"):
      if temp_estop_var_vention=="estop/status true":
      sendStringWithTimeout("estop/systemreset/request","Ack estop/systemreset/request;","MachineMotion1")
      end
      socket_send_string("estop/status;", "MachineMotion1")
      temp_estop_var_vention = socket_read_string("MachineMotion1",timeout=15)
      if temp_estop_var_vention=="estop/status true":
      popup("MachineMotion in estop, make sure you have all emergency modules released manually. If you continue the system will try to reset MachineMotion automatically.",blocking=True)
      end
      end
      else:
      popup("resource is being used already: MachineMotion1")
      halt
      end
      isVentionMovementBusyMachineMotion1 = True
      sendString("im_home_axis_1", "MachineMotion im_home_axis_1 = completed", "MachineMotion1")
      isVentionMovementBusyMachineMotion1 = False
      sendString("SET im_set_encoder_pos_aux_1 0.000", "Ack", "MachineMotion1")
      isVentionMovementBusyMachineMotion1 = False
      sleep(0.03)
      # end: URCap Program Node
    end
    $ 342 "'now go into the ccw weld position'"
    # 'now go into the ccw weld position'
    $ 343 "Waypoint_29" "breakAfter"
    movej(get_inverse_kin(Waypoint_29_p, qnear=Waypoint_29_q), a=1.3962634015954636, v=1.3962634015954636)
    $ 344 "Comment"
    # Comment
    $ 345 "Waypoint_30" "breakAfter"
    movej(get_inverse_kin(Waypoint_30_p, qnear=Waypoint_30_q), a=1.3962634015954636, v=1.3962634015954636)
    $ 346 "Waypoint_31" "breakAfter"
    movej(get_inverse_kin(Waypoint_31_p, qnear=Waypoint_31_q), a=1.3962634015954636, v=1.3962634015954636)
    $ 355 "MoveL"
    $ 356 "p_pre_ret" "breakAfter"
    movel(p_pre_ret, a=1.2, v=0.25)
    $ 357 "p_pre_ret2" "breakAfter"
    movel(p_pre_ret2, a=1.2, v=0.25)
    $ 358 "p_preheat" "breakAfter"
    movel(p_preheat, a=1.2, v=0.25)
    $ 359 "Wait: 6.0"
    sleep(6.0)
    $ 360 "MoveL"
    $ 361 "p_pre_ret2" "breakAfter"
    movel(p_pre_ret2, a=1.2, v=0.25)
    $ 362 "p_pre_ret" "breakAfter"
    movel(p_pre_ret, a=1.2, v=0.25)
    $ 363 "Set"
    set_tcp(p[0.00451,-0.328,0.105,1.2092,-1.2092,1.2092])
    $ 364 "MoveL"
    $ 365 "p_1" "breakAfter"
    movel(p_1, a=0.1, v=0.05)
    # begin: URCap Program Node
    #   Source: WireTank Serial, 4.9.0, WireTank, LLC
    #   Type: WireTank Serial
    $ 366 "Serial Bridge uR1"
    SerialResponse = WTSerialBridge.send_command("/dev/ttyUSB0",1200, 8, "None", "One", "None", 1000, "None", "None", [252,82,49], False)
    # end: URCap Program Node
    # begin: URCap Program Node
    #   Source: WireTank Serial, 4.9.0, WireTank, LLC
    #   Type: WireTank Serial
    $ 367 "Serial Bridge uR1"
    SerialResponse = WTSerialBridge.send_command("/dev/ttyUSB0",1200, 8, "None", "One", "None", 1000, "None", "None", [252,82,49], False)
    # end: URCap Program Node
    $ 368 "Wait: 1.0"
    sleep(1.0)
    $ 369 "Set DO[0]=On"
    set_standard_digital_out(0, True)
    $ 371 "Wait: 1.0"
    sleep(1.0)
    $ 372 "MoveL"
    $ 373 "p_2" "breakAfter"
    movel(p_2, a=1.2, v=0.01)
    $ 374 "MoveP"
    $ 375 "CircleMove"
    $ 376 "p_3" "noBreak"

    $ 377 "p_4" "breakAfter"
    movec(p_3, p_4, a=0.01, v=5.0E-4, r=0.0, mode=1)
    $ 378 "MoveL"
    $ 379 "p_5" "breakAfter"
    movel(p_5, a=1.2, v=0.012)
    $ 380 "Set"
    set_tcp(p[-0.011699999999999999,-0.328,0.105,1.2092,-1.2092,1.2092])
    $ 381 "MoveL"
    $ 382 "p_6" "breakAfter"
    movel(p_6, a=0.1, v=0.012)
    $ 383 "p_7" "breakAfter"
    movel(p_7, a=0.1, v=0.012)
    # begin: URCap Program Node
    #   Source: WireTank Serial, 4.9.0, WireTank, LLC
    #   Type: WireTank Serial
    $ 384 "Serial Bridge uR0"
    SerialResponse = WTSerialBridge.send_command("/dev/ttyUSB0",1200, 8, "None", "One", "None", 1000, "None", "None", [252,82,48], False)
    # end: URCap Program Node
    $ 386 "Set DO[0]=Off"
    set_standard_digital_out(0, False)
    $ 387 "MoveL"
    $ 388 "p_8" "breakAfter"
    movel(p_8, a=0.1, v=0.01)
    $ 389 "Set DO[0]=Off"
    set_standard_digital_out(0, False)
    $ 394 "MoveJ"
    $ 395 "Waypoint_32" "breakAfter"
    movej(get_inverse_kin(Waypoint_32_p, qnear=Waypoint_32_q), a=1.3962634015954636, v=1.0471975511965976)
    $ 396 "Waypoint_33" "breakAfter"
    movej(get_inverse_kin(Waypoint_33_p, qnear=Waypoint_33_q), a=1.3962634015954636, v=1.0471975511965976)
    $ 397 "Waypoint_73" "breakAfter"
    movej(get_inverse_kin(Waypoint_73_p, qnear=Waypoint_73_q), a=1.3962634015954636, v=1.0471975511965976)
    $ 398 "Comment"
    # Comment
    $ 399 "MoveJ"
    $ 400 "Waypoint_16" "breakAfter"
    movej(get_inverse_kin(Waypoint_16_p, qnear=Waypoint_16_q), a=1.3962634015954636, v=1.0471975511965976)
    $ 401 "Waypoint_17" "breakAfter"
    movej(get_inverse_kin(Waypoint_17_p, qnear=Waypoint_17_q), a=1.3962634015954636, v=1.0471975511965976)
    $ 402 "Waypoint_18" "breakAfter"
    movej(get_inverse_kin(Waypoint_18_p, qnear=Waypoint_18_q), a=1.3962634015954636, v=1.0471975511965976)
    $ 403 "Waypoint_38" "breakAfter"
    movej(get_inverse_kin(Waypoint_38_p, qnear=Waypoint_38_q), a=1.3962634015954636, v=1.0471975511965976)
    $ 404 "'above point is home'"
    # 'above point is home'
  end
  def Test_Teach_Position():
    $ 405 "Test_Teach_Position" "noBreak"
    $ 409 "MoveJ"
    $ 410 "Waypoint_40" "breakAfter"
    set_tcp(p[0.0,0.0,0.019,0.0,0.0,0.0])
    movej(get_inverse_kin(Waypoint_40_p, qnear=Waypoint_40_q), a=1.3962634015954636, v=1.0471975511965976)
    $ 411 "'above waypoint is home'"
    # 'above waypoint is home'
    $ 412 "Waypoint_2" "breakAfter"
    set_tcp(p[0.0,0.0,0.019,0.0,0.0,0.0])
    movej(get_inverse_kin(Waypoint_2_p, qnear=Waypoint_2_q), a=1.3962634015954636, v=1.0471975511965976)
    $ 413 "Set"
    set_tcp(p[1.4000000000000001E-4,-0.01751,0.285,0.0,0.0,0.0])
    $ 414 "freedrive_m_var≔ False "
    global freedrive_m_var=  False
    $ 415 "freedrive_m_var≔ True "
    global freedrive_m_var=  True
    $ 416 "Popup: Move the TCP to the top of the weld, then click 'Continue'"
    popup("Move the TCP to the top of the weld, then click 'Continue'", "Message", False, False, blocking=True)
    $ 417 "tcp_pose_top≔get_actual_tcp_pose()"
    global tcp_pose_top= get_actual_tcp_pose ()
    $ 418 "Popup: Move the TCP to the corner of the tank, then click 'Continue'"
    popup("Move the TCP to the corner of the tank, then click 'Continue'", "Message", False, False, blocking=True)
    $ 419 "tcp_pose≔get_actual_tcp_pose()"
    global tcp_pose= get_actual_tcp_pose ()
    $ 420 "freedrive_m_var≔ False "
    global freedrive_m_var=  False
    $ 421 "Wait: 0.25"
    sleep(0.25)
    $ 422 "sync()"
    sync()
  end
  def align_tcp_left():
    $ 423 "align_tcp_left" "noBreak"
    $ 424 "'this program aligns the tcp parallel to the y direction'"
    # 'this program aligns the tcp parallel to the y direction'
    $ 425 "cp≔get_actual_tcp_pose()"
    global cp= get_actual_tcp_pose ()
    $ 426 "aligned_y_pose≔p[cp[0],cp[1],cp[2],1.570796,0,0]"
    global aligned_y_pose=p[cp[0],cp[1],cp[2],1.570796,0,0]
    $ 427 "MoveJ"
    $ 428 "aligned_y_pose" "breakAfter"
    movej(aligned_y_pose, a=1.3962634015954636, v=1.0471975511965976)
  end
  def extrude_knife3():
    $ 429 "extrude_knife3" "noBreak"
    $ 430 "pre program stuff"
    $ 431 "Set"
    set_tcp(p[-0.011699999999999999,-0.328,0.105,1.2092,-1.2092,1.2092])
    $ 432 "ek_sp≔get_actual_tcp_pose()"
    global ek_sp= get_actual_tcp_pose ()
    $ 433 "MoveL"
    $ 434 "ek_sp" "breakAfter"
    movel(ek_sp, a=1.2, v=0.005)
    $ 435 "'list possible points'"
    # 'list possible points'
    $ 436 "robot 1 moves"
    $ 437 "If 1≟2"
    if (1 == 2):
      $ 438 "MoveJ"
      $ 439 "r1_ek_oldhome" "breakAfter"
      movej(get_inverse_kin(r1_ek_oldhome_p, qnear=r1_ek_oldhome_q), a=1.3962634015954636, v=1.0471975511965976)
      $ 440 "r1_ek_extrude" "breakAfter"
      movej(get_inverse_kin(r1_ek_extrude_p, qnear=r1_ek_extrude_q), a=1.3962634015954636, v=1.0471975511965976)
      $ 441 "r1_ek_front" "breakAfter"
      movej(get_inverse_kin(r1_ek_front_p, qnear=r1_ek_front_q), a=1.3962634015954636, v=1.0471975511965976)
      $ 442 "r1_ek_middle" "breakAfter"
      movej(get_inverse_kin(r1_ek_middle_p, qnear=r1_ek_middle_q), a=1.3962634015954636, v=1.0471975511965976)
      $ 443 "r1_ek_middle2" "breakAfter"
      movej(get_inverse_kin(r1_ek_middle2_p, qnear=r1_ek_middle2_q), a=1.3962634015954636, v=1.0471975511965976)
      $ 444 "r1_ek_bottom" "breakAfter"
      movej(get_inverse_kin(r1_ek_bottom_p, qnear=r1_ek_bottom_q), a=1.3962634015954636, v=1.0471975511965976)
      $ 445 "r1_ek_end" "breakAfter"
      movej(get_inverse_kin(r1_ek_end_p, qnear=r1_ek_end_q), a=1.3962634015954636, v=1.0471975511965976)
    end
    $ 446 "robot 2 moves"
    $ 447 "If 1≟2"
    if (1 == 2):
      $ 448 "MoveJ"
      $ 449 "r2_ek_oldhome" "breakAfter"
      movej(get_inverse_kin(r2_ek_oldhome_p, qnear=r2_ek_oldhome_q), a=1.3962634015954636, v=1.0471975511965976)
      $ 451 "r2_ek_extrude" "breakAfter"
      movej(get_inverse_kin(r2_ek_extrude_p, qnear=r2_ek_extrude_q), a=1.3962634015954636, v=1.0471975511965976)
      $ 452 "r2_ek_front" "breakAfter"
      movej(get_inverse_kin(r2_ek_front_p, qnear=r2_ek_front_q), a=1.3962634015954636, v=1.0471975511965976)
      $ 453 "r2_ek_middle" "breakAfter"
      movej(get_inverse_kin(r2_ek_middle_p, qnear=r2_ek_middle_q), a=1.3962634015954636, v=1.0471975511965976)
      $ 454 "r2_ek_bottom" "breakAfter"
      movej(get_inverse_kin(r2_ek_bottom_p, qnear=r2_ek_bottom_q), a=1.3962634015954636, v=1.0471975511965976)
      $ 455 "r2_ek_end" "breakAfter"
      movej(get_inverse_kin(r2_ek_end_p, qnear=r2_ek_end_q), a=1.3962634015954636, v=1.0471975511965976)
    end
    $ 456 "robot 3 moves"
    $ 457 "If 1≟2"
    if (1 == 2):
      $ 458 "MoveJ"
      $ 459 "r3_ek_oldhome" "breakAfter"
      movej(get_inverse_kin(r3_ek_oldhome_p, qnear=r3_ek_oldhome_q), a=1.3962634015954636, v=1.0471975511965976)
      $ 460 "r3_ek_extrude" "breakAfter"
      movej(get_inverse_kin(r3_ek_extrude_p, qnear=r3_ek_extrude_q), a=1.3962634015954636, v=1.0471975511965976)
      $ 461 "r3_ek_front" "breakAfter"
      movej(get_inverse_kin(r3_ek_front_p, qnear=r3_ek_front_q), a=1.3962634015954636, v=1.0471975511965976)
      $ 462 "r3_ek_middle" "breakAfter"
      movej(get_inverse_kin(r3_ek_middle_p, qnear=r3_ek_middle_q), a=1.3962634015954636, v=1.0471975511965976)
      $ 463 "r3_ek_bottom" "breakAfter"
      movej(get_inverse_kin(r3_ek_bottom_p, qnear=r3_ek_bottom_q), a=1.3962634015954636, v=1.0471975511965976)
      $ 464 "r3_ek_end" "breakAfter"
      movej(get_inverse_kin(r3_ek_end_p, qnear=r3_ek_end_q), a=1.3962634015954636, v=1.0471975511965976)
    end
    $ 465 "robot 4 moves"
    $ 466 "If 1≟2"
    if (1 == 2):
      $ 467 "MoveJ"
      $ 468 "r4_ek_oldhome" "breakAfter"
      movej(get_inverse_kin(r4_ek_oldhome_p, qnear=r4_ek_oldhome_q), a=1.3962634015954636, v=1.0471975511965976)
      $ 469 "r4_ek_extrude" "breakAfter"
      movej(get_inverse_kin(r4_ek_extrude_p, qnear=r4_ek_extrude_q), a=1.3962634015954636, v=1.0471975511965976)
      $ 470 "r4_ek_front" "breakAfter"
      movej(get_inverse_kin(r4_ek_front_p, qnear=r4_ek_front_q), a=1.3962634015954636, v=1.0471975511965976)
      $ 471 "r4_ek_middle" "breakAfter"
      movej(get_inverse_kin(r4_ek_middle_p, qnear=r4_ek_middle_q), a=1.3962634015954636, v=1.0471975511965976)
      $ 472 "r4_ek_bottom" "breakAfter"
      movej(get_inverse_kin(r4_ek_bottom_p, qnear=r4_ek_bottom_q), a=1.3962634015954636, v=1.0471975511965976)
      $ 473 "r4_ek_end" "breakAfter"
      movej(get_inverse_kin(r4_ek_end_p, qnear=r4_ek_end_q), a=1.3962634015954636, v=1.0471975511965976)
    end
    $ 474 "'detemine correct points for which robot'"
    # 'detemine correct points for which robot'
    $ 475 "If robot_number≟1"
    if (robot_number == 1):
      $ 476 "robot1 positions"
      $ 477 "ek_oldhome≔r1_ek_oldhome_p"
      global ek_oldhome=r1_ek_oldhome_p
      $ 478 "ek_extrude≔r1_ek_extrude_p"
      global ek_extrude=r1_ek_extrude_p
      $ 479 "ek_front≔r1_ek_front_p"
      global ek_front=r1_ek_front_p
      $ 480 "ek_middle≔r1_ek_middle_p"
      global ek_middle=r1_ek_middle_p
      $ 481 "ek_middle2≔r1_ek_middle2_p"
      global ek_middle2=r1_ek_middle2_p
      $ 482 "ek_bottom≔r1_ek_bottom_p"
      global ek_bottom=r1_ek_bottom_p
      $ 483 "ek_end≔r1_ek_end_q"
      global ek_end=r1_ek_end_q
    else:
      $ 484 "ElseIf robot_number≟2"
      if (robot_number == 2):
        $ 485 "robot2 positions"
        $ 486 "ek_oldhome≔r2_ek_oldhome_p"
        global ek_oldhome=r2_ek_oldhome_p
        $ 487 "ek_extrude≔r2_ek_extrude_p"
        global ek_extrude=r2_ek_extrude_p
        $ 488 "ek_front≔r2_ek_front_p"
        global ek_front=r2_ek_front_p
        $ 489 "ek_middle≔r2_ek_middle_p"
        global ek_middle=r2_ek_middle_p
        $ 490 "ek_middle2≔r2_ek_middle_p"
        global ek_middle2=r2_ek_middle_p
        $ 491 "ek_bottom≔r2_ek_bottom_p"
        global ek_bottom=r2_ek_bottom_p
        $ 492 "ek_end≔r2_ek_end_q"
        global ek_end=r2_ek_end_q
      else:
        $ 493 "ElseIf robot_number≟3"
        if (robot_number == 3):
          $ 494 "robot3 positions"
          $ 495 "ek_oldhome≔r3_ek_oldhome_p"
          global ek_oldhome=r3_ek_oldhome_p
          $ 496 "ek_extrude≔r3_ek_extrude_p"
          global ek_extrude=r3_ek_extrude_p
          $ 497 "ek_front≔r3_ek_front_p"
          global ek_front=r3_ek_front_p
          $ 498 "ek_middle≔r3_ek_middle_p"
          global ek_middle=r3_ek_middle_p
          $ 499 "ek_middle2≔r3_ek_middle_p"
          global ek_middle2=r3_ek_middle_p
          $ 500 "ek_bottom≔r3_ek_bottom_p"
          global ek_bottom=r3_ek_bottom_p
          $ 501 "ek_end≔r3_ek_end_q"
          global ek_end=r3_ek_end_q
        else:
          $ 502 "ElseIf robot_number≟4"
          if (robot_number == 4):
            $ 503 "robot4 positions"
            $ 504 "ek_oldhome≔r4_ek_oldhome_p"
            global ek_oldhome=r4_ek_oldhome_p
            $ 505 "ek_extrude≔r4_ek_extrude_p"
            global ek_extrude=r4_ek_extrude_p
            $ 506 "ek_front≔r4_ek_front_p"
            global ek_front=r4_ek_front_p
            $ 507 "ek_middle≔r4_ek_middle_p"
            global ek_middle=r4_ek_middle_p
            $ 508 "ek_middle2≔r4_ek_middle_p"
            global ek_middle2=r4_ek_middle_p
            $ 509 "ek_bottom≔r4_ek_bottom_p"
            global ek_bottom=r4_ek_bottom_p
            $ 510 "ek_end≔r4_ek_end_q"
            global ek_end=r4_ek_end_q
          end
        end
      end
    end
    $ 511 "'start of program'"
    # 'start of program'
    $ 513 "Set"
    set_tcp(p[-0.011699999999999999,-0.328,0.105,1.2092,-1.2092,1.2092])
    $ 514 "MoveJ"
    $ 516 "ek_oldhome" "breakAfter"
    movej(ek_oldhome, a=1.3962634015954636, v=1.0471975511965976)
    $ 517 "'above waypoint is home'"
    # 'above waypoint is home'
    $ 518 "'move above bucket'"
    # 'move above bucket'
    $ 519 "MoveJ"
    $ 521 "ek_extrude" "breakAfter"
    movej(ek_extrude, a=1.3962634015954636, v=1.0471975511965976)
    $ 522 "'extrude out a foot'"
    # 'extrude out a foot'
    # begin: URCap Program Node
    #   Source: WireTank Serial, 4.9.0, WireTank, LLC
    #   Type: WireTank Serial
    $ 524 "Serial Bridge uR1"
    SerialResponse = WTSerialBridge.send_command("/dev/ttyUSB0",1200, 8, "None", "One", "None", 1000, "None", "None", [252,82,49], False)
    # end: URCap Program Node
    $ 525 "Set DO[0]=On"
    set_standard_digital_out(0, True)
    $ 526 "Wait: 24.0"
    sleep(24.0)
    # begin: URCap Program Node
    #   Source: WireTank Serial, 4.9.0, WireTank, LLC
    #   Type: WireTank Serial
    $ 527 "Serial Bridge uR0"
    SerialResponse = WTSerialBridge.send_command("/dev/ttyUSB0",1200, 8, "None", "One", "None", 1000, "None", "None", [252,82,48], False)
    # end: URCap Program Node
    $ 528 "Wait: 1.0"
    sleep(1.0)
    $ 529 "Set DO[0]=Off"
    set_standard_digital_out(0, False)
    $ 530 "'slice'"
    # 'slice'
    $ 531 "MoveL"
    $ 537 "ek_front" "breakAfter"
    movel(ek_front, a=0.05, v=0.03)
    $ 538 "ek_middle" "breakAfter"
    movel(ek_middle, a=0.05, v=0.03)
    $ 539 "ek_middle2" "breakAfter"
    movel(ek_middle2, a=0.05, v=0.03)
    $ 540 "ek_bottom" "breakAfter"
    movel(ek_bottom, a=0.05, v=0.03)
    $ 541 "ek_end" "breakAfter"
    movel(ek_end, a=0.05, v=0.03)
    $ 542 "MoveJ"
    $ 544 "ek_oldhome" "breakAfter"
    movej(ek_oldhome, a=1.3962634015954636, v=1.0471975511965976)
    $ 545 "'above waypoint is home'"
    # 'above waypoint is home'
  end
  def align_tcp_forward():
    $ 547 "align_tcp_forward" "noBreak"
    $ 548 "'this program aligns the tcp parallel to the y direction'"
    # 'this program aligns the tcp parallel to the y direction'
    $ 549 "cp≔get_actual_tcp_pose()"
    global cp= get_actual_tcp_pose ()
    $ 550 "aligned_y_pose≔p[cp[0],cp[1],cp[2],0,-1.570796,0]"
    global aligned_y_pose=p[cp[0],cp[1],cp[2],0,-1.570796,0]
    $ 551 "MoveJ"
    $ 552 "aligned_y_pose" "breakAfter"
    movej(aligned_y_pose, a=1.3962634015954636, v=1.0471975511965976)
  end
  def align_tcp_up():
    $ 553 "align_tcp_up" "noBreak"
    $ 554 "'this program aligns the tcp parallel to the y direction'"
    # 'this program aligns the tcp parallel to the y direction'
    $ 555 "cp≔get_actual_tcp_pose()"
    global cp= get_actual_tcp_pose ()
    $ 556 "aligned_y_pose≔p[cp[0],cp[1],cp[2],0,0,0]"
    global aligned_y_pose=p[cp[0],cp[1],cp[2],0,0,0]
    $ 557 "MoveJ"
    $ 558 "aligned_y_pose" "breakAfter"
    movej(aligned_y_pose, a=1.3962634015954636, v=1.0471975511965976)
  end
  def align_ready_for_welding():
    $ 559 "align_ready_for_welding" "noBreak"
    $ 560 "'this program takes the welder from home to a position alined ready for welding (vertically down)'"
    # 'this program takes the welder from home to a position alined ready for welding (vertically down)'
    $ 561 "MoveJ"
    $ 562 "oldhome" "breakAfter"
    movej(get_inverse_kin(oldhome_p, qnear=oldhome_q), a=1.3962634015954636, v=1.0471975511965976)
    $ 563 "Waypoint_34" "breakAfter"
    movej(get_inverse_kin(Waypoint_34_p, qnear=Waypoint_34_q), a=1.3962634015954636, v=1.0471975511965976)
    $ 564 "Waypoint_35" "breakAfter"
    movej(get_inverse_kin(Waypoint_35_p, qnear=Waypoint_35_q), a=1.3962634015954636, v=1.0471975511965976)
    $ 565 "Waypoint_36" "breakAfter"
    movej(get_inverse_kin(Waypoint_36_p, qnear=Waypoint_36_q), a=1.3962634015954636, v=1.0471975511965976)
  end
  def Corner_Homing_45():
    $ 566 "Corner_Homing_45" "noBreak"
    $ 567 "'Use this program when tool is already positioned close to corner at 45deg'"
    # 'Use this program when tool is already positioned close to corner at 45deg'
    $ 568 "'tool flange will seek all 3 sides. will save those 5 locs in p__'"
    # 'tool flange will seek all 3 sides. will save those 5 locs in p__'
    $ 569 "Set"
    set_tcp(p[1.4000000000000001E-4,-0.01751,0.285,0.0,0.0,0.0])
    $ 578 "Wait: 1.0"
    sleep(1.0)
    $ 579 "tp≔get_actual_tcp_pose()"
    global tp= get_actual_tcp_pose ()
    $ 583 "path_pre≔get_corner_homing_45_pathpoints(tp,tcp_pose_top)"
    global path_pre=get_corner_homing_45_pathpoints(tp,tcp_pose_top)
    $ 584 "ph1≔path_pre[0]"
    global ph1=path_pre[0]
    $ 585 "ph2≔path_pre[1]"
    global ph2=path_pre[1]
    $ 586 "ph3≔path_pre[2]"
    global ph3=path_pre[2]
    $ 587 "ph4≔path_pre[3]"
    global ph4=path_pre[3]
    $ 588 "ph5≔path_pre[4]"
    global ph5=path_pre[4]
    $ 589 "ph6≔path_pre[5]"
    global ph6=path_pre[5]
    $ 590 "ph7≔path_pre[6]"
    global ph7=path_pre[6]
    $ 591 "ph2up≔path_pre[7]"
    global ph2up=path_pre[7]
    $ 592 "ph4up≔path_pre[8]"
    global ph4up=path_pre[8]
    $ 593 "MoveL"
    $ 594 "ph1" "breakAfter"
    movel(ph1, a=0.2, v=0.25)
    $ 595 "ph2" "breakAfter"
    movel(ph2, a=0.2, v=0.25)
    $ 596 "Wait: 0.5"
    sleep(0.5)
    $ 597 "MoveL"
    $ 598 "Direction: Base"
    global move_thread_flag_598=0
    thread move_thread_598():
      enter_critical
      move_thread_flag_598 = 1
      local towardsPos=calculate_point_to_move_towards(p[0.0,0.0,0.0,0.0,0.0,0.0], [-1,-1.0,0.0], 1000.0)
      movel(towardsPos, a=0.1, v=0.02)
      move_thread_flag_598 = 2
      exit_critical
    end
    move_thread_flag_598 = 0
    move_thread_han_598 = run move_thread_598()
    while (True):
      local targetTcpDirection=get_target_tcp_speed()
      local stepsToRetract=tool_contact(direction=targetTcpDirection)
      if (stepsToRetract > 0):
        kill move_thread_han_598
        stopl(3.0)
        local backTrackMovement=get_actual_joint_positions_history(stepsToRetract)
        local contactPose=get_forward_kin(backTrackMovement)
        local posDir=[targetTcpDirection[0],targetTcpDirection[1],targetTcpDirection[2]]
        local retractTo=contactPose
        if (norm(posDir) > 1e-6):
          local normalizedPosDir=normalize(posDir)
          local additionalRetraction=p[normalizedPosDir[0] * 0.0, normalizedPosDir[1] * 0.0, normalizedPosDir[2] * 0.0, 0, 0, 0]
          retractTo = pose_sub(contactPose, additionalRetraction)
        end
        movel(retractTo, a=3.0, v=0.1)
        $ 599 "Until (tool_contact_detection)"
        break
      end
      sync()
    end
    $ 600 "p11≔get_actual_tcp_pose()"
    global p11= get_actual_tcp_pose ()
    $ 601 "MoveJ"
    $ 602 "ph2" "breakAfter"
    movej(ph2, a=1.3962634015954636, v=1.0471975511965976)
    $ 603 "ph2up" "breakAfter"
    movej(ph2up, a=1.3962634015954636, v=1.0471975511965976)
    $ 604 "Wait: 0.5"
    sleep(0.5)
    $ 605 "MoveL"
    $ 606 "Direction: Base"
    global move_thread_flag_606=0
    thread move_thread_606():
      enter_critical
      move_thread_flag_606 = 1
      local towardsPos=calculate_point_to_move_towards(p[0.0,0.0,0.0,0.0,0.0,0.0], [-1,-1.0,0.0], 1000.0)
      movel(towardsPos, a=0.1, v=0.02)
      move_thread_flag_606 = 2
      exit_critical
    end
    move_thread_flag_606 = 0
    move_thread_han_606 = run move_thread_606()
    while (True):
      local targetTcpDirection=get_target_tcp_speed()
      local stepsToRetract=tool_contact(direction=targetTcpDirection)
      if (stepsToRetract > 0):
        kill move_thread_han_606
        stopl(3.0)
        local backTrackMovement=get_actual_joint_positions_history(stepsToRetract)
        local contactPose=get_forward_kin(backTrackMovement)
        local posDir=[targetTcpDirection[0],targetTcpDirection[1],targetTcpDirection[2]]
        local retractTo=contactPose
        if (norm(posDir) > 1e-6):
          local normalizedPosDir=normalize(posDir)
          local additionalRetraction=p[normalizedPosDir[0] * 0.0, normalizedPosDir[1] * 0.0, normalizedPosDir[2] * 0.0, 0, 0, 0]
          retractTo = pose_sub(contactPose, additionalRetraction)
        end
        movel(retractTo, a=3.0, v=0.1)
        $ 607 "Until (tool_contact_detection)"
        break
      end
      sync()
    end
    $ 608 "p13≔get_actual_tcp_pose()"
    global p13= get_actual_tcp_pose ()
    $ 609 "MoveJ"
    $ 610 "ph2up" "breakAfter"
    movej(ph2up, a=1.3962634015954636, v=1.0471975511965976)
    $ 611 "ph3" "breakAfter"
    movej(ph3, a=1.3962634015954636, v=1.0471975511965976)
    $ 612 "Wait: 0.5"
    sleep(0.5)
    $ 613 "MoveL"
    $ 614 "Direction: Base"
    global move_thread_flag_614=0
    thread move_thread_614():
      enter_critical
      move_thread_flag_614 = 1
      local towardsPos=calculate_point_to_move_towards(p[0.0,0.0,0.0,0.0,0.0,0.0], [-1,-1.0,0.0], 1000.0)
      movel(towardsPos, a=0.1, v=0.02)
      move_thread_flag_614 = 2
      exit_critical
    end
    move_thread_flag_614 = 0
    move_thread_han_614 = run move_thread_614()
    while (True):
      local targetTcpDirection=get_target_tcp_speed()
      local stepsToRetract=tool_contact(direction=targetTcpDirection)
      if (stepsToRetract > 0):
        kill move_thread_han_614
        stopl(3.0)
        local backTrackMovement=get_actual_joint_positions_history(stepsToRetract)
        local contactPose=get_forward_kin(backTrackMovement)
        local posDir=[targetTcpDirection[0],targetTcpDirection[1],targetTcpDirection[2]]
        local retractTo=contactPose
        if (norm(posDir) > 1e-6):
          local normalizedPosDir=normalize(posDir)
          local additionalRetraction=p[normalizedPosDir[0] * 0.0, normalizedPosDir[1] * 0.0, normalizedPosDir[2] * 0.0, 0, 0, 0]
          retractTo = pose_sub(contactPose, additionalRetraction)
        end
        movel(retractTo, a=3.0, v=0.1)
        $ 615 "Until (tool_contact_detection)"
        break
      end
      sync()
    end
    $ 616 "p12≔get_actual_tcp_pose()"
    global p12= get_actual_tcp_pose ()
    $ 620 "MoveL"
    $ 621 "ph3" "breakAfter"
    movel(ph3, a=1.2, v=0.25)
    $ 622 "ph1" "breakAfter"
    movel(ph1, a=1.2, v=0.25)
    $ 627 "MoveL"
    $ 628 "ph4" "breakAfter"
    movel(ph4, a=1.2, v=0.25)
    $ 629 "Wait: 0.5"
    sleep(0.5)
    $ 630 "MoveL"
    $ 631 "Direction: Base"
    global move_thread_flag_631=0
    thread move_thread_631():
      enter_critical
      move_thread_flag_631 = 1
      local towardsPos=calculate_point_to_move_towards(p[0.0,0.0,0.0,0.0,0.0,0.0], [-1.0,1.0,0.0], 1000.0)
      movel(towardsPos, a=0.1, v=0.02)
      move_thread_flag_631 = 2
      exit_critical
    end
    move_thread_flag_631 = 0
    move_thread_han_631 = run move_thread_631()
    while (True):
      local targetTcpDirection=get_target_tcp_speed()
      local stepsToRetract=tool_contact(direction=targetTcpDirection)
      if (stepsToRetract > 0):
        kill move_thread_han_631
        stopl(3.0)
        local backTrackMovement=get_actual_joint_positions_history(stepsToRetract)
        local contactPose=get_forward_kin(backTrackMovement)
        local posDir=[targetTcpDirection[0],targetTcpDirection[1],targetTcpDirection[2]]
        local retractTo=contactPose
        if (norm(posDir) > 1e-6):
          local normalizedPosDir=normalize(posDir)
          local additionalRetraction=p[normalizedPosDir[0] * 0.0, normalizedPosDir[1] * 0.0, normalizedPosDir[2] * 0.0, 0, 0, 0]
          retractTo = pose_sub(contactPose, additionalRetraction)
        end
        movel(retractTo, a=3.0, v=0.1)
        $ 632 "Until (tool_contact_detection)"
        break
      end
      sync()
    end
    $ 633 "p21≔get_actual_tcp_pose()"
    global p21= get_actual_tcp_pose ()
    $ 634 "MoveL"
    $ 635 "ph4" "breakAfter"
    movel(ph4, a=1.2, v=0.25)
    $ 636 "ph4up" "breakAfter"
    movel(ph4up, a=1.2, v=0.25)
    $ 637 "Wait: 0.5"
    sleep(0.5)
    $ 638 "MoveL"
    $ 639 "Direction: Base"
    global move_thread_flag_639=0
    thread move_thread_639():
      enter_critical
      move_thread_flag_639 = 1
      local towardsPos=calculate_point_to_move_towards(p[0.0,0.0,0.0,0.0,0.0,0.0], [-1.0,1.0,0.0], 1000.0)
      movel(towardsPos, a=0.1, v=0.02)
      move_thread_flag_639 = 2
      exit_critical
    end
    move_thread_flag_639 = 0
    move_thread_han_639 = run move_thread_639()
    while (True):
      local targetTcpDirection=get_target_tcp_speed()
      local stepsToRetract=tool_contact(direction=targetTcpDirection)
      if (stepsToRetract > 0):
        kill move_thread_han_639
        stopl(3.0)
        local backTrackMovement=get_actual_joint_positions_history(stepsToRetract)
        local contactPose=get_forward_kin(backTrackMovement)
        local posDir=[targetTcpDirection[0],targetTcpDirection[1],targetTcpDirection[2]]
        local retractTo=contactPose
        if (norm(posDir) > 1e-6):
          local normalizedPosDir=normalize(posDir)
          local additionalRetraction=p[normalizedPosDir[0] * 0.0, normalizedPosDir[1] * 0.0, normalizedPosDir[2] * 0.0, 0, 0, 0]
          retractTo = pose_sub(contactPose, additionalRetraction)
        end
        movel(retractTo, a=3.0, v=0.1)
        $ 640 "Until (tool_contact_detection)"
        break
      end
      sync()
    end
    $ 641 "p23≔get_actual_tcp_pose()"
    global p23= get_actual_tcp_pose ()
    $ 642 "MoveL"
    $ 643 "ph4up" "breakAfter"
    movel(ph4up, a=1.2, v=0.25)
    $ 644 "ph5" "breakAfter"
    movel(ph5, a=1.2, v=0.25)
    $ 645 "Wait: 0.5"
    sleep(0.5)
    $ 646 "MoveL"
    $ 647 "Direction: Base"
    global move_thread_flag_647=0
    thread move_thread_647():
      enter_critical
      move_thread_flag_647 = 1
      local towardsPos=calculate_point_to_move_towards(p[0.0,0.0,0.0,0.0,0.0,0.0], [-1.0,1.0,0.0], 1000.0)
      movel(towardsPos, a=0.1, v=0.02)
      move_thread_flag_647 = 2
      exit_critical
    end
    move_thread_flag_647 = 0
    move_thread_han_647 = run move_thread_647()
    while (True):
      local targetTcpDirection=get_target_tcp_speed()
      local stepsToRetract=tool_contact(direction=targetTcpDirection)
      if (stepsToRetract > 0):
        kill move_thread_han_647
        stopl(3.0)
        local backTrackMovement=get_actual_joint_positions_history(stepsToRetract)
        local contactPose=get_forward_kin(backTrackMovement)
        local posDir=[targetTcpDirection[0],targetTcpDirection[1],targetTcpDirection[2]]
        local retractTo=contactPose
        if (norm(posDir) > 1e-6):
          local normalizedPosDir=normalize(posDir)
          local additionalRetraction=p[normalizedPosDir[0] * 0.0, normalizedPosDir[1] * 0.0, normalizedPosDir[2] * 0.0, 0, 0, 0]
          retractTo = pose_sub(contactPose, additionalRetraction)
        end
        movel(retractTo, a=3.0, v=0.1)
        $ 648 "Until (tool_contact_detection)"
        break
      end
      sync()
    end
    $ 649 "p22≔get_actual_tcp_pose()"
    global p22= get_actual_tcp_pose ()
    $ 660 "MoveJ"
    $ 661 "ph5" "breakAfter"
    movej(ph5, a=1.3962634015954636, v=1.0471975511965976)
    $ 662 "MoveL"
    $ 663 "ph4" "breakAfter"
    movel(ph4, a=1.2, v=0.25)
    $ 664 "ph1" "breakAfter"
    movel(ph1, a=1.2, v=0.25)
    $ 665 "MoveJ"
    $ 666 "Waypoint_4" "breakAfter"
    movej(get_inverse_kin(Waypoint_4_p, qnear=Waypoint_4_q), a=1.3962634015954636, v=1.0471975511965976)
    $ 667 "Waypoint_13" "breakAfter"
    movej(get_inverse_kin(Waypoint_13_p, qnear=Waypoint_13_q), a=1.3962634015954636, v=1.0471975511965976)
    $ 668 "Waypoint_1" "breakAfter"
    movej(get_inverse_kin(Waypoint_1_p, qnear=Waypoint_1_q), a=1.3962634015954636, v=1.0471975511965976)
    $ 669 "ph6" "breakAfter"
    movej(ph6, a=1.3962634015954636, v=1.0471975511965976)
    $ 670 "ph7" "breakAfter"
    movej(ph7, a=1.3962634015954636, v=1.0471975511965976)
    $ 671 "Wait: 1.0"
    sleep(1.0)
    $ 675 "MoveL"
    $ 676 "Direction: Base Z+"
    global move_thread_flag_676=0
    thread move_thread_676():
      enter_critical
      move_thread_flag_676 = 1
      local towardsPos=calculate_point_to_move_towards(p[0.0,0.0,0.0,0.0,0.0,0.0], [0.0,0.0,1.0], 1000.0)
      movel(towardsPos, a=0.1, v=0.02)
      move_thread_flag_676 = 2
      exit_critical
    end
    move_thread_flag_676 = 0
    move_thread_han_676 = run move_thread_676()
    while (True):
      local targetTcpDirection=get_target_tcp_speed()
      local stepsToRetract=tool_contact(direction=targetTcpDirection)
      if (stepsToRetract > 0):
        kill move_thread_han_676
        stopl(3.0)
        local backTrackMovement=get_actual_joint_positions_history(stepsToRetract)
        local contactPose=get_forward_kin(backTrackMovement)
        local posDir=[targetTcpDirection[0],targetTcpDirection[1],targetTcpDirection[2]]
        local retractTo=contactPose
        if (norm(posDir) > 1e-6):
          local normalizedPosDir=normalize(posDir)
          local additionalRetraction=p[normalizedPosDir[0] * 0.0, normalizedPosDir[1] * 0.0, normalizedPosDir[2] * 0.0, 0, 0, 0]
          retractTo = pose_sub(contactPose, additionalRetraction)
        end
        movel(retractTo, a=3.0, v=0.1)
        $ 677 "Until (tool_contact_detection)"
        break
      end
      sync()
    end
    $ 678 "p3≔get_actual_tcp_pose()"
    global p3= get_actual_tcp_pose ()
    $ 679 "MoveJ"
    $ 680 "ph7" "breakAfter"
    movej(ph7, a=1.3962634015954636, v=1.0471975511965976)
    $ 681 "ph6" "breakAfter"
    movej(ph6, a=1.3962634015954636, v=1.0471975511965976)
    $ 682 "Waypoint_14" "breakAfter"
    movej(get_inverse_kin(Waypoint_14_p, qnear=Waypoint_14_q), a=1.3962634015954636, v=1.0471975511965976)
    $ 683 "Waypoint_4" "breakAfter"
    movej(get_inverse_kin(Waypoint_4_p, qnear=Waypoint_4_q), a=1.3962634015954636, v=1.0471975511965976)
    $ 684 "Waypoint_41" "breakAfter"
    movej(get_inverse_kin(Waypoint_41_p, qnear=Waypoint_41_q), a=1.3962634015954636, v=1.0471975511965976)
    $ 685 "'above waypoint is home'"
    # 'above waypoint is home'
    $ 687 "Comment"
    # Comment
    $ 688 "Comment"
    # Comment
    $ 689 "Comment"
    # Comment
    $ 690 "Comment"
    # Comment
    $ 691 "Comment"
    # Comment
    $ 692 "Comment"
    # Comment
  end
  $ 2 "BeforeStart"
  $ 3 "Safe Home Folder"
  $ 4 "'if robot is not at home, send it back to home safely'"
  # 'if robot is not at home, send it back to home safely'
  $ 5 "'make sure the tcp is welder'"
  # 'make sure the tcp is welder'
  $ 6 "Set"
  set_tcp(p[-0.011699999999999999,-0.328,0.105,1.2092,-1.2092,1.2092])
  $ 7 "sp≔get_actual_tcp_pose()"
  global sp= get_actual_tcp_pose ()
  $ 8 "MoveL"
  $ 9 "sp" "breakAfter"
  movel(sp, a=1.2, v=0.25)
  $ 10 "'if first move is to a variable, skip automove'"
  # 'if first move is to a variable, skip automove'
  $ 11 "'turn off welder'"
  # 'turn off welder'
  # begin: URCap Program Node
  #   Source: WireTank Serial, 4.9.0, WireTank, LLC
  #   Type: WireTank Serial
  $ 12 "Serial Bridge uR0"
  SerialResponse = WTSerialBridge.send_command("/dev/ttyUSB0",1200, 8, "None", "One", "None", 1000, "None", "None", [252,82,48], False)
  # end: URCap Program Node
  $ 13 "Set DO[0]=Off"
  set_standard_digital_out(0, False)
  $ 14 "jp≔get_actual_joint_positions()"
  global jp= get_actual_joint_positions ()
  $ 15 "If sp[0]>0.600"
  if (sp[0]>0.600):
    $ 16 "'if x > 600 then above then home'"
    # 'if x > 600 then above then home'
    $ 17 "MoveJ"
    $ 19 "Waypoint_76" "breakAfter"
    movej(get_inverse_kin(Waypoint_76_p, qnear=Waypoint_76_q), a=1.3962634015954636, v=1.0471975511965976)
    $ 20 "Home"
    movej([-3.266929759358355, -1.2139462677784536, 1.5878387874396154, 1.1069165929565088, -0.0023738326664366483, -1.7891447305770605], a=1.3962634015954636, v=1.0471975511965976)
  else:
    $ 21 "Else" "noBreak"
    $ 22 "Popup: retreating to home"
    popup("retreating to home", "Message", False, False, blocking=True)
    $ 23 "'for rules 2-8, finish with oldhome then above then home'"
    # 'for rules 2-8, finish with oldhome then above then home'
    $ 24 "If -1.74<jp[4] and jp[4]<1.05 and -1.74<jp[3] and jp[3]<1.74"
    if (-1.74<jp[4]  and  jp[4]<1.05  and  -1.74<jp[3]  and  jp[3]<1.74):
      $ 25 "'if oldhome, test teach, then go straight to oldhome'"
      # 'if oldhome, test teach, then go straight to oldhome'
    else:
      $ 26 "ElseIf sp[0]<-.5 and jp[3]>3.14 and -2.62<jp[4] and jp[4]<-0.87"
      if (sp[0]<-.5  and  jp[3]>3.14  and  -2.62<jp[4]  and  jp[4]<-0.87):
        $ 27 "'if left side weld approach, left weld approach in reverse'"
        # 'if left side weld approach, left weld approach in reverse'
        $ 28 "MoveJ"
        $ 29 "Waypoint_50" "breakAfter"
        movej(get_inverse_kin(Waypoint_50_p, qnear=Waypoint_50_q), a=1.3962634015954636, v=1.0471975511965976)
        $ 30 "Waypoint_51" "breakAfter"
        movej(get_inverse_kin(Waypoint_51_p, qnear=Waypoint_51_q), a=1.3962634015954636, v=1.0471975511965976)
        $ 31 "Waypoint_52" "breakAfter"
        movej(get_inverse_kin(Waypoint_52_p, qnear=Waypoint_52_q), a=1.3962634015954636, v=1.0471975511965976)
        $ 32 "Waypoint_53" "breakAfter"
        movej(get_inverse_kin(Waypoint_53_p, qnear=Waypoint_53_q), a=1.3962634015954636, v=1.0471975511965976)
      else:
        $ 33 "ElseIf sp[0]<0 and 0<jp[3] and jp[3]<1.74 and 0.87<jp[4] and jp[4]<2.62"
        if (sp[0]<0  and  0<jp[3]  and  jp[3]<1.74  and  0.87<jp[4]  and  jp[4]<2.62):
          $ 34 "'if right side around, move back then wapoint 24 then oldhome'"
          # 'if right side around, move back then wapoint 24 then oldhome'
          $ 35 "If sp[0]<-1.0"
          if (sp[0]<-1.0):
            $ 36 "xback≔p[-1.0,sp[1],sp[2],sp[3],sp[4],sp[5]]"
            global xback=p[-1.0,sp[1],sp[2],sp[3],sp[4],sp[5]]
            $ 37 "MoveJ"
            $ 38 "xback" "breakAfter"
            movej(xback, a=1.3962634015954636, v=1.0471975511965976)
          end
          $ 39 "MoveJ"
          $ 40 "Waypoint_54" "breakAfter"
          movej(get_inverse_kin(Waypoint_54_p, qnear=Waypoint_54_q), a=1.3962634015954636, v=1.0471975511965976)
        else:
          $ 41 "ElseIf jp[3]>2.62 and jp[4]<-3.84"
          if (jp[3]>2.62  and  jp[4]<-3.84):
            $ 42 "'if left side second half, then left weld ending sequence'"
            # 'if left side second half, then left weld ending sequence'
            $ 43 "If jp[5]<0.35"
            if (jp[5]<0.35):
              $ 44 "MoveJ"
              $ 45 "Waypoint_65" "breakAfter"
              movej(get_inverse_kin(Waypoint_65_p, qnear=Waypoint_65_q), a=1.3962634015954636, v=1.0471975511965976)
            end
            $ 46 "MoveJ"
            $ 51 "'above is testing, below is real'"
            # 'above is testing, below is real'
            $ 52 "Waypoint_55" "breakAfter"
            movej(get_inverse_kin(Waypoint_55_p, qnear=Waypoint_55_q), a=1.3962634015954636, v=1.0471975511965976)
            $ 54 "Waypoint_59" "breakAfter"
            movej(get_inverse_kin(Waypoint_59_p, qnear=Waypoint_59_q), t=2.0)
            $ 55 "Waypoint_71" "breakAfter"
            movej(get_inverse_kin(Waypoint_71_p, qnear=Waypoint_71_q), a=1.3962634015954636, v=1.0471975511965976)
            $ 56 "Waypoint_58" "breakAfter"
            movej(get_inverse_kin(Waypoint_58_p, qnear=Waypoint_58_q), a=1.3962634015954636, v=1.0471975511965976)
            $ 57 "Waypoint_56" "breakAfter"
            movej(get_inverse_kin(Waypoint_56_p, qnear=Waypoint_56_q), a=1.3962634015954636, v=1.0471975511965976)
            $ 58 "Waypoint_57" "breakAfter"
            movej(get_inverse_kin(Waypoint_57_p, qnear=Waypoint_57_q), a=1.3962634015954636, v=1.0471975511965976)
          else:
            $ 59 "ElseIf jp[3]<-2.09"
            if (jp[3]<-2.09):
              $ 60 "'bottom homing'"
              # 'bottom homing'
              $ 61 "MoveJ"
              $ 63 "Comment"
              # Comment
              $ 64 "If sp[0]<-0.95"
              if (sp[0]<-0.95):
                $ 65 "xback≔p[-0.95,sp[1],sp[2],sp[3],sp[4],sp[5]]"
                global xback=p[-0.95,sp[1],sp[2],sp[3],sp[4],sp[5]]
                $ 66 "MoveL"
                $ 67 "xback" "breakAfter"
                movel(xback, a=1.2, v=0.25)
              end
              $ 68 "Waypoint_67" "breakAfter"
              movej(get_inverse_kin(Waypoint_67_p, qnear=Waypoint_67_q), a=1.3962634015954636, v=1.0471975511965976)
            else:
              $ 69 "ElseIf jp[3]<0 and jp[4]<-3.14"
              if (jp[3]<0  and  jp[4]<-3.14):
                $ 70 "'if left side homing, special unspin'"
                # 'if left side homing, special unspin'
                $ 71 "MoveJ"
                $ 73 "Comment"
                # Comment
                $ 74 "Waypoint_69" "breakAfter"
                movej(get_inverse_kin(Waypoint_69_p, qnear=Waypoint_69_q), a=1.3962634015954636, v=1.0471975511965976)
                $ 75 "Waypoint_70" "breakAfter"
                movej(get_inverse_kin(Waypoint_70_p, qnear=Waypoint_70_q), a=1.3962634015954636, v=1.0471975511965976)
              else:
                $ 76 "ElseIf (sp[4]<-3 or sp[4]>3) and -0.02<sp[5] and sp[5]<0.02"
                if ((sp[4]<-3  or  sp[4]>3)  and  -0.02<sp[5]  and  sp[5]<0.02):
                  $ 77 "'go straight to home'"
                  # 'go straight to home'
                else:
                  $ 78 "ElseIf 2>1"
                  if (2>1):
                    $ 79 "'if none of the other options, then error continuously'"
                    # 'if none of the other options, then error continuously'
                    $ 80 "Loop 2>1"
                    while (2>1):
                      $ 81 "Popup: Unknown Position. Find Calvin for Assistance"
                      popup("Unknown Position. Find Calvin for Assistance", "Message", False, False, blocking=True)
                    end
                  end
                end
              end
            end
          end
        end
      end
    end
    $ 82 "'insert logic for how to get back to oldhome'"
    # 'insert logic for how to get back to oldhome'
    $ 83 "'finish with oldhome then above then home'"
    # 'finish with oldhome then above then home'
    $ 84 "MoveJ"
    $ 85 "Waypoint_49" "breakAfter"
    movej(get_inverse_kin(Waypoint_49_p, qnear=Waypoint_49_q), a=1.3962634015954636, v=1.0471975511965976)
    $ 87 "Waypoint_75" "breakAfter"
    movej(get_inverse_kin(Waypoint_75_p, qnear=Waypoint_75_q), a=1.3962634015954636, v=1.0471975511965976)
    $ 88 "Home"
    movej([-3.266929759358355, -1.2139462677784536, 1.5878387874396154, 1.1069165929565088, -0.0023738326664366483, -1.7891447305770605], a=1.3962634015954636, v=1.0471975511965976)
    # begin: URCap Program Node
    #   Source: MachineLogic for Universal Robots, 3.1.7, Vention Inc.
    #   Type: MachineLogic for Universal Robots
    $ 89 "MachineLogic Homing"
    while isVentionMovementBusyMachineMotion1==True:
    sleep(0.05)
    end
    if(isVentionMovementBusyMachineMotion1 == False):
    isVentionMovementBusyMachineMotion1 = True
    socket_send_string("estop/status;", "MachineMotion1")
    temp_estop_var_vention = socket_read_string("MachineMotion1",timeout=15)
    while(temp_estop_var_vention=="estop/status true"):
    if temp_estop_var_vention=="estop/status true":
    sendStringWithTimeout("estop/systemreset/request","Ack estop/systemreset/request;","MachineMotion1")
    end
    socket_send_string("estop/status;", "MachineMotion1")
    temp_estop_var_vention = socket_read_string("MachineMotion1",timeout=15)
    if temp_estop_var_vention=="estop/status true":
    popup("MachineMotion in estop, make sure you have all emergency modules released manually. If you continue the system will try to reset MachineMotion automatically.",blocking=True)
    end
    end
    else:
    popup("resource is being used already: MachineMotion1")
    halt
    end
    isVentionMovementBusyMachineMotion1 = True
    sendString("im_home_axis_1", "MachineMotion im_home_axis_1 = completed", "MachineMotion1")
    isVentionMovementBusyMachineMotion1 = False
    sendString("SET im_set_encoder_pos_aux_1 0.000", "Ack", "MachineMotion1")
    isVentionMovementBusyMachineMotion1 = False
    sleep(0.03)
    # end: URCap Program Node
  end
  $ 693 "Thread_1"
  thread Thread_1():
    $ 694 "Loop  True "
    while (  True  ):
      $ 695 "If freedrive_m_var≟ True "
      if (freedrive_m_var ==   True  ):
        $ 696 "freedrive_mode()"
        freedrive_mode()
        $ 697 "free_dr_already≔ True "
        global free_dr_already=  True
      else:
        $ 698 "Else" "noBreak"
        $ 699 "If free_dr_already"
        if (free_dr_already):
          $ 700 "end_freedrive_mode()"
          end_freedrive_mode()
        end
      end
      $ 701 "sync()"
      sync()
    end
  end
  threadId_Thread_1 = run Thread_1()
  $ 90 "Robot Program"
  $ 91 "'start of main program'"
  # 'start of main program'
  $ 92 "Set"
  set_tcp(p[-0.011699999999999999,-0.328,0.105,1.2092,-1.2092,1.2092])
  $ 93 "Home"
  movej([-3.266929759358355, -1.2139462677784536, 1.5878387874396154, 1.1069165929565088, -0.0023738326664366483, -1.7891447305770605], a=1.3962634015954636, v=1.0471975511965976)
  $ 94 "Script: common_math.script"
  # define pi
  pi = 3.1415926535

  # given 3 points, this finds the plane and its equation
  # rereturns ax + by + cz + d = 0 in a list of [a, b, c, d]
  def findplane(p11, p12, p13):
      # extract coordinates
      x1 = p11[0]
      y1 = p11[1]
      z1 = p11[2]
      x2 = p12[0]
      y2 = p12[1]
      z2 = p12[2]
      x3 = p13[0]
      y3 = p13[1]
      z3 = p13[2]
      # create vectors from the points
      v1x = x2-x1
      v1y = y2-y1
      v1z = z2-z1
      v2x = x3-x1
      v2y = y3-y1
      v2z = z3-z1
      #calculate the normal vector using the cross product
      nx = v1y*v2z - v1z*v2y # i component
      ny = v1z*v2x - v1x*v2z # j component
      nz = v1x*v2y - v1y*v2x # k component
      # calculate d in the plane equation
      d = -1 * (nx*x1 + ny*y1 + nz*z1)
      ret = [nx, ny, nz, d]
      return ret
  end

  # given a heading, (ccw from +x axis), find the mx+b slope
  # fails if exactly vertical
  def get_slope_from_heading(heading):
      return tan(heading)
  end

  # this function converts a unit vector to its heading angle ccw from x+ axis
  # takes uvx and uvy
  # returns heading in radians
  def convert_uv_to_heading(uvx, uvy):
    baseang = atan(uvy/uvx)
    if uvx < 0:
      ang = baseang + pi
    elif uvy < 0:
      ang = baseang + pi * 2
    else:
      ang = baseang
    end
    return ang
  end

  # this function finds the equation of a line, perpendicular to a given line, and going through a given point
  # takes 3 arguments: m (the original line's slope), x (point's x coord), y (point's y coord). the b of the original line is not needed
  # returns a list of [m,b] (the slope and intercept of the new line)
  def find_perpendicular_line(origm, x, y):
    m = (1/origm) * -1
    b = y - m*x
    ret = [m, b]
    return ret
  end

  # this function finds the intersection point between two lines in the xy plane
  # takes 4 arguments: m1, b1, m2, b2
  # returns a list of [x,y] (the point of intersection)
  def find_intersection(m1, b1, m2, b2):
    # m1x+b1 = m2x+b2
    # m1x - m2x = b2 - b1
    # x = (b2-b1) / (m1-m2)
    x = (b2-b1) / (m1-m2)
    y = m1 * x + b1
    ret = [x, y]
    return ret
  end

  # this function finds the distance between 2 points in 3d space
  # it takes 6 arguments: x1, y1, z1, x2, y2, z2
  # it returns a distance
  def distance_between(x1, y1, z1, x2, y2, z2):
    distsquared = (x2-x1)*(x2-x1)+(y2-y1)*(y2-y1)+(z2-z1)*(z2-z1)
    dist = sqrt(distsquared)
    return dist
  end

  # this function takes a point, a unit vector, and a distance, and adds the distance to the point in the direction of the unit vector (3d space)
  # it returns a point as a list of coordinates
  def add_vectordistance_to_point(xi, yi, zi, uvx, uvy, uvz, delta):
    xf = xi + uvx * delta
    yf = yi + uvy * delta
    zf = zi + uvz * delta
    ret = [xf, yf, zf]
    return ret
  end

  # this function converts a heading (ccw radians from the positive x axis) into rxryrz to be put into a point p[]
  # this will point the gun in this heading with the bottom side of the gun facing up.
  # the values used in this program were calculated by doing rotation matrix math in the file on WI-CALVINB10 C. Documents. Theory for converting rotations into axis angle representations
  def convert_heading_to_axang(heading):
   axisxraw = -1 * sin(heading)
   axisyraw = cos(heading) + 1
   axiszraw = sin(heading)

   magnitude = sqrt(axisxraw*axisxraw + axisyraw*axisyraw + axiszraw*axiszraw)

   axisxunit = axisxraw / magnitude
   axisyunit = axisyraw / magnitude
   axiszunit = axiszraw / magnitude

   angle = acos( (cos(heading) - 1) / 2 )

   rxout = axisxunit * angle
   ryout = axisyunit * angle
   rzout = axiszunit * angle

   return [rxout, ryout, rzout]
  end

  # this function converts a heading (ccw radians from the positive x axis) into rxryrz to be put into a point p[]
  # this will point the gun in this heading with the preheat side of the gun tip facing up. Used for welding in a vertical path.
  # the values used in this program were calculated by doing rotation matrix math in the file on WI-CALVINB10 C. Documents. Theory for converting rotations into axis angle representations
  def convert_heading_to_axang_preheatup(heading):
   axisxraw = -sin(heading) + 1
   axisyraw = cos(heading)
   axiszraw = cos(heading)

   magnitude = sqrt(axisxraw*axisxraw + axisyraw*axisyraw + axiszraw*axiszraw)

   axisxunit = axisxraw / magnitude
   axisyunit = axisyraw / magnitude
   axiszunit = axiszraw / magnitude

   angle = acos( (-sin(heading) - 1) / 2 )

   rxout = axisxunit * angle
   ryout = axisyunit * angle
   rzout = axiszunit * angle

   return [rxout, ryout, rzout]
  end

  # this function converts a heading (ccw radians from the positive x axis) into rxryrz to be put into a point p[]
  # this will point the gun in this heading with the preheat side of the gun tip facing down. Used for welding in a vertical path downwards.
  # the values used in this program were calculated by doing rotation matrix math in the file on WI-CALVINB10 C. Documents. Theory for converting rotations into axis angle representations
  def convert_heading_to_axang_preheatdown(heading):
   axisxraw = -sin(heading) - 1
   axisyraw = cos(heading)
   axiszraw = -cos(heading)

   magnitude = sqrt(axisxraw*axisxraw + axisyraw*axisyraw + axiszraw*axiszraw)

   axisxunit = axisxraw / magnitude
   axisyunit = axisyraw / magnitude
   axiszunit = axiszraw / magnitude

   angle = acos( (sin(heading) - 1) / 2 )

   rxout = axisxunit * angle
   ryout = axisyunit * angle
   rzout = axiszunit * angle

   return [rxout, ryout, rzout]
  end

  # this function converts a heading (ccw radians from the positive x axis) into rxryrz to be put into a point p[]
  # this will point the gun in this heading with the preheat side of the gun tip facing right. Used for welding counterclockwise around the box.
  # the values used in this program were calculated by doing rotation matrix math in the file on WI-CALVINB10 C. Documents. Theory for converting rotations into axis angle representations
  def convert_heading_to_axang_ccw(heading):
   axisxraw = -sin(heading)
   axisyraw = cos(heading) - 1
   axiszraw = -sin(heading)

   magnitude = sqrt(axisxraw*axisxraw + axisyraw*axisyraw + axiszraw*axiszraw)

   axisxunit = axisxraw / magnitude
   axisyunit = axisyraw / magnitude
   axiszunit = axiszraw / magnitude

   angle = acos( (-cos(heading) - 1) / 2 )

   rxout = axisxunit * angle
   ryout = axisyunit * angle
   rzout = axiszunit * angle

   return [rxout, ryout, rzout]
  end

